	// GRID
		CmdAutCpl					: BOOL; 		(* Coupling authorization	*)
		CmdDisconnect				: BOOL; 		(* Powerplant disconnect order *)
		CmdEmergencyDisconnect		: BOOL; 		(* Powerplant Emergency disconnect order *)
		
	//Project specific ( France ) 
	CmdDisconnect_end			: BOOL; 		(* Powerplant End of disconnect order *)
	CmdEmergencyDisconnect_end	: BOOL; 		(* Powerplant End of Emergency disconnect order *)
	CmdStartPReg				: BOOL ; 		(* Activate P regulation from Grid   *)
	CmdStopPreg                 : BOOL ; 		(* Desactivate P regulation from Grid   *)
	CmdStartQReg                : BOOL ; 		(* Activate Q regulation from Grid   *)
	CmdStopQReg                 : BOOL ; 		(* Desactivate Q regulation from Grid   *)

           	
END_STRUCT
END_TYPE

// ---- 04_Application/OPC/AllDataWToggle.TcDUT
TYPE AllDataWToggle :
STRUCT
	// Toggle command
		CmdStopServer_SMS		: BOOL ;	(* Disable SMS Server *)
		
END_STRUCT
END_TYPE

// ---- 04_Application/OPC/AllValueW.TcDUT
TYPE AllValueW :
STRUCT
 // PP 
	SetptTanPhi_PP				: REAL; 										(* (p.u) TanPhi setpoint to regulate if the corresponding mode is activated *)

// SMS 	
	AX_NbPhone_OPC				: ARRAY[1..CstNbUser] OF STRING(26);			(* List of the phone number to be registered for SMS functions *)
	AX_SubscribedSms_OPC		: ARRAY[1..CstNbUser] OF BOOL;					(* List of subscription for SMS function *)
	AX_NamesUsers_OPC					: ARRAY[1..CstNbUser] OF STRING(50);	(* List of SMS user names *)
	AX_MailAddr_OPC				: ARRAY[1..CstNbUser] OF STRING(255);			(* Contient tous les numéros des utilisateurs *)
	AX_SubscribedMail_OPC		: ARRAY[1..CstNbUser] OF BOOL;					(* List of subscription for MAIL function *)
	AX_UserLVL					: ARRAY[1..CstNbUser] OF WORD;					(* Bit-wise encoding of Alarm subscription (Check Config alarm document for bit signification) *)
	
// SUB	
	SetpP_SUB					: REAL;											(* (kW) Active Power setpoint to be regulated at Subatstion ( if local setpoint enabled) *)
    SetpQ_SUB					: REAL;											(* (kVAr) Reactive Power setpoint to be regulated at Subatstion ( if local setpoint enabled) *)
// PTR 
	SetpP_INV					: ARRAY[1..CstNbPTR_G] OF ARRAY[1..CstNbInv_PTR_G] OF  REAL;	(*(kW) Active Power setpoint to be regulated at the inverter ( if local setpoint enabled) *) 	
	
END_STRUCT
END_TYPE

// ---- 00_FunctionsBlocks/Beckhoff/Communication/IEC104/GVL_Cst.TcGVL
{attribute 'qualified_only'}
VAR_GLOBAL CONSTANT
		CstNbAOEntries			: INT :=  50 ;
END_VAR

// ---- 00_FunctionsBlocks/Beckhoff/Fifo/GVL_Fifo.TcGVL
VAR_GLOBAL CONSTANT 
		Max_buffer_size_G					: UDINT:=10000000; // Max buffer size of fifo
END_VAR

// ---- 04_Application/CONFIG/GVL_BASE.TcGVL
///////////////////////
// DO NOT MODIFY :  
// Maximal number of objects  - Maximal array size 
////////////////////
VAR_GLOBAL CONSTANT 
	// PRODUCT 
	CstNbPTR_G					: BYTE := 4 ;  				// (NA) Number of PTR
	CstNbESS_G   				: BYTE := 3 ;  				// (NA) Number of ESS


// EQUIPMENT
	
	//SUB_MV
	
		CstNbFeederMVCB_G			: BYTE	:= 3 ; 
		CstNbGridMVCB_G				: BYTE	:= 2 ; 
	
	// PTR 
	
		CstNbInv_PTR_G				: BYTE := 5 ;	// Maximal Number of PV Inverters for PTR
		CstNbTempTansfo_PTR_G		: BYTE := 2 ; 	// Maximal Number of Transformer temperature
		CstNbSB_INV_G				: BYTE := 32 ;	// Maximal Number of String box in inverter
		CstNb_DU_G					: BYTE := 2  ;	// Maximal number of DU ? DC inputs ? 
		CstNbPowerCol_INV_G			: BYTE := 3 ; 	// Maximal number of Power Columns per inverter 
		CstNbSB_DcModule_G			: BYTE := 15 ; 	// Maximal number of String box in DC Module 
		CstNbDcModule_INV_G			: BYTE := 15 ;	 // Maximal number of DC Module by inverter
		CstNbSTR_SB_G				: BYTE := 32 ;	// Maximal Number of String by String box 
		
	// EM 
		
		CstNbEM_G					: BYTE := 2;				// Number of Energy Meters
		
	//ESS		
	
		CstNbPcs_ESS_G					: BYTE := 2  ;
		CstNbPowerCol_PCS_G				: BYTE := 6  ;				// Maximal Number of Power colonne by PCS
		CstNbHvac_ESS_G					: BYTE := 2  ;
		CstNbBAT_ESS_G					: BYTE := 2  ;
		CstNbRack_BAT_G					: BYTE := 2  ;
		CstNbModule_Rack_G				: BYTE := 25  ;
		CstNbBms_BAT_G					: BYTE := 1  ;
		CstNbDU_PCS_G					: BYTE := 2  ;
		CstNbTempSensor_ESS_G			: BYTE := 4  ;
		CstNbHygroSensor_ESS_G			: BYTE := 4  ;
		CstNbDS_Ess_G					: BYTE := 2  ;
		CstNbSS_Ess_G					: BYTE := 2  ;
		CstNbEs_ESS_G					: BYTE := 2  ;
		CstNbChainDcSwitchBank_Ess_G	: BYTE := 2  ;	
		
		
	//WS	
	
		CstNbPyrano_GTI				: UINT := 5;
		CstNbPyrano_GHI				: UINT := 5;
		CstNbAnemo					: UINT := 1;
		CstNbPanTmp					: UINT := 4;
		CstNbAmbTmp					: UINT := 3;	
		
	// PP 
	
		CstNbCouplermax_G			: BYTE 	:= 100 ;			// Maximal number of ethercat devices 
		CstNbAlarmIO_G				: BYTE := 10 ; // Number of Event in PRG_IO.
		
	//TRK 
	
		CstNbTrk_NCU_G				: BYTE := 200 ; 
	
	(*               SMS               							*)
	CstNbUser					: SINT:=10; //Nbr d'utilisateur utilisé par AX_Numtel
	CstNbCMD					: SINT:=20; //Nbr commande utilisé par AX_CMD_SMS
	CstNbAlarmCode				: INT:=400;  //Number of alarmcode use in AlarmManager
	
	// TIMEZONE
	    (* Indonesia East Standard Time Zone settings *)
        FRANCE_TZI : ST_TimeZoneInformation := (bias:=-60,
                                       		 				standardName:='Heure Française',
                                        					standardDate:=(wYear:=0,wMonth:=10,wDayOfWeek:=0,wDay:=27,wHour:=3),
                                        					standardBias:=0,
                                        					daylightName:='None',
                                        					daylightDate:=(wYear:=0,wMonth:=3,wDayOfWeek:=0,wDay:=31,wHour:=2),
                                        					daylightBias:=0);
			
		CstPhoneIndicator_G		: STRING := '+33';
			
			CstCycleTime_G		: INT := 10 ; 			// (ms) Cycle Time of the CPU FB Main 
			CstCycleTime_Annex	: INT := 100 ; 			// (ms) Cycle Time of the CPU FB Annex_Function

		CstNbRedundantVariableMax_G	: UINT := 553 ;
		CstNbParamOPCUA				: UINT := 100 ; 
	
END_VAR
VAR_GLOBAL
	sTimeGMT_G          	: STRING;				// Full Date Time for historization (GMT) 
	sTimeLocal_G		 	: STRING ;				// Local Time 
	CalGMTTimeStruct		: TIMESTRUCT ; 			// GMT Time Structure

	ParamOpenVpnFile		: STRING := '';			// Path to openvpn file. 
	ParamIpPublic 			: STRING(255);			// Public IP 
	MesSizeCdrive_PLC		: REAL := 100000 ; 		// (Mo) Remaining Disk space
	MesSizeCdrive_IndusPC	: REAL := 100000 ; 		// (Mo) Remaining Disk space
END_VAR

// ---- 04_Application/CONFIG/GVL_Beckhoff.TcGVL
VAR_GLOBAL
	CalLocalTimeStruct			: TIMESTRUCT;		// Local Time Structure
	CstTimeZone_G				: ST_TimeZoneInformation 	:= WEST_EUROPE_TZI ;	// Local TimeZone
	ParamDirBaseStore		: STRING := 'C:\TwinCAT\Functions\Historisation\';	// Directroy for the historization
	
	
	// Communication 
	stPCComInData  	AT %I*	: EL6inData22B;//PcComInData; 	//DATA qui rentre  ELinData22B;
	stPCComOutData	AT %Q*	: El6outdata22b;//PcComOutData; //DATA qui sort  EL6outData22B;
	stTxBufferPC			: ComBuffer; 	//Connection serie
	stRxBufferPC			: ComBuffer; 	//Connection serie
	
END_VAR

// ---- 04_Application/CONFIG/GVL_CFG.TcGVL
///////////////
// Configuration Files. Define Power Plant sizing and references. 
//////////////
VAR_GLOBAL 
		CstPLCBackup 			: BOOL := FALSE ;  			// TRUE if this PLC is used as a backup . 
		CstNetAmsId_Slave		: STRING(20):= '5.49.202.22.1.1'; //NetAMSId Slave .'5.79.170.90.1.1'
		CstNetAmsId_IndusPC		: STRING(20):= ''; // set '' if no Indus PLC
		//CstIPIEC104			: STRING := '10.101.111.1' ; 
		
		
END_VAR
	
VAR_GLOBAL 
	// Solar Classique //
		A1_PP					: FB_PP  ;  								// MCA Power Plant 
 
	// PRODUCT DEFINITION //
		//PTR 
		AX_PTR 					: ARRAY[1..CstNbPTR_G] OF FB_PTR ; 	 		// Array with AMG products
		
		//SUB_MV
		A1_SUBMV				: FB_SUBMV ;	 					 		// SUB_MV		

		//SUB_HV
		A1_SUBHV				: FB_SUBHV ;	 					 		// SUB_MV		


		
		//WEATHER STATION
		A1_WS					: FB_WS;
		
		//ESS 
		AX_ESS				: ARRAY[1..CstNbESS_G] OF FB_ESS ; 
		
	// GLOBAL VARIABLE //
	
		CmdClearFault_G			: BOOL ; 									// (NA) Clear all permanent faults
		CmdInit_G				: BOOL ; 									// (NA) Global Init Action
		CstIPIEC104				: STRING := '10.111.109.1' ; 		
END_VAR

// ---- 04_Application/CONFIG/GVL_Check.TcGVL
VAR_GLOBAL
	FaultCheck_G : BOOL ; // Test if Fault 
	Fault_Count_G: CTU  ; // Counter 	
	

END_VAR

// ---- 04_Application/CONFIG/GVL_DataBaseStructures.TcGVL
{attribute 'qualified_only'}
VAR_GLOBAL
	AX_StructModbusTCP 	AT %MW112 	: ARRAY[1..10000] OF WORD;
END_VAR

// ---- 04_Application/Annexes_Functions/PRG_AnnexesFunctions.TcPOU
PROGRAM PRG_AnnexesFunctions
VAR_INPUT PERSISTENT
	ParamServiceName_OPCUA			: STRING(255) := 'OPCUA\';	(*OPC UA Folder Name*)
	ParamServiceName_Teamviewer		: STRING(255) := 'Teamviewer\';	(* Teamviewer Folder Name*)	
	ParamServiceName_HMIServer		: STRING(255) := 'HmiServer\';	(*HmiServer Service Name*)	
	ParamServiceName_Telegraf		: STRING(255) := 'Telegraf\';	(* Telegraf Folder Name*)	
END_VAR
VAR_INPUT
	IN_bStartPing				: BOOL;	
    IN_bStart_IP				: BOOL;
    IN_bStart_PLC				: BOOL;

	IN_CmdRestart_OPCUA 		: BOOL;	// OPC UA , Docker , OPEn VPN , Codesys. Push button
	IN_CmdRestart_Teamviewer 	: BOOL;	// OPC UA , Docker , OPEn VPN , Codesys. Push button
	IN_CmdRestart_HMIServer 	: BOOL;	// OPC UA , Docker , OPEn VPN , Codesys. Push button
	IN_CmdRestart_Telegraf 		: BOOL;	// OPC UA , Docker , OPEn VPN , Codesys. Push button

	IN_bStartVpnConnection		: BOOL;
	IN_bStopVpnConnection		: BOOL;
	IN_AdrIP					: STRING(50);
END_VAR

VAR_INPUT PERSISTENT
	ParamRestartTCHour			: WORD := 3;
	ParamRestartTCEnabled		: BOOL ; 
END_VAR

VAR PERSISTENT 
	RestartCounter 				: UINT;
END_VAR

VAR
		bInit					: BOOL := TRUE ; 
		PRG_RestartService		: ARRAY[1..4] OF FB_RestartService ; 
		StartProcess 			: NT_StartProcess;
		CpuUsage				: TC_CpuUsage;
		TON_ALarm				: TON ; // TON to inhibate alarmes during the first secondes after initailization 

		// Restart Twincta
		Step: INT;
		R_Trig_TP_IP			: R_TRIG;
		TC_Restart1				: TC_Restart;	
		TP_GetIPPublic			: TP;

END_VAR
VAR_OUTPUT 
	CPUUsage_PLC				: UDINT ; 
END_VAR

IF bInit THEN
	M_Init();
	///////// 
END_IF




// Get Public IP : 	Auto query every 10 minutes
	FUN_GetPublicIp(
		ParamNetID := CstNetAmsId_IndusPC ,
		IN_DirExe := 'C:\TwinCAT\Functions\Annex_Fonctions\GetPublicIp\',
		IN_CmdStart := IN_bStart_IP OR (CalLocalTimeStruct.wMinute MOD 10 = 0 AND CalLocalTimeStruct.wSecond = 0
	));

// Ping Host 	
//	FUN_PingHost(IN_bStart := IN_bStartPing, IN_PingAdr := IN_AdrIP, IN_DirBatLocation := 'C:\TwinCAT\Functions\Fonction_Com\Ping\');

// CHECK STATES
	// CPU Usage 	
		CpuUsage(NETID := '', Start := CalLocalTimeStruct.wSecond = 0, TMOUT := T#1S);
		CPUUsage_PLC := 	CpuUsage.USAGE ; 
		
	// Check Disk Space = planned task
	// Check Services = planned task
	// Network Scan = planned task
	
	// VPN Management
		FUN_ConnectVPN(IN_CmdStart := IN_bStartVpnConnection, IN_OpenVpnFile := GVL_BASE.ParamOpenVpnFile);
		FUN_DisconnectVPN(IN_CmdStart := IN_bStopVpnConnection);
		

// RESTART SERVICES 
	// Restart OPC UA  	


			PRG_RestartService[1](ParamNetID:='' , IN_Directory := CONCAT(STR1:='C:\TwinCAT\Functions\AnnexFunctions\RestartService\',STR2:= ParamServiceName_OPCUA), Start:= IN_CmdRestart_OPCUA , IN_ServiceName := 'RestartService.exe');
			PRG_RestartService[2](ParamNetID:='' , IN_Directory := CONCAT(STR1:='C:\TwinCAT\Functions\AnnexFunctions\RestartService\',STR2:= ParamServiceName_Teamviewer), Start:= IN_CmdRestart_Teamviewer , IN_ServiceName := 'RestartService.exe');
			PRG_RestartService[3](ParamNetID:='' , IN_Directory := CONCAT(STR1:='C:\TwinCAT\Functions\AnnexFunctions\RestartService\',STR2:= ParamServiceName_HMIServer), Start:= IN_CmdRestart_HMIServer , IN_ServiceName := 'RestartService.exe');
			PRG_RestartService[4](ParamNetID:='' , IN_Directory := CONCAT(STR1:='C:\TwinCAT\Functions\AnnexFunctions\RestartService\',STR2:= ParamServiceName_Telegraf), Start:= IN_CmdRestart_Telegraf , IN_ServiceName := 'RestartService.exe');



	// Restart PLC 	
		PRG_RestartPlc(CmdRestart:= IN_bStart_PLC);
		
	// Restart Twincat at specified date and time to fix EL6614 issue 
		CASE Step OF
			0: //	
				IF CalLocalTimeStruct.wHour = ParamRestartTCHour AND CalLocalTimeStruct.wMinute = 0 AND (CalLocalTimeStruct.wSecond >= 0 AND CalLocalTimeStruct.wSecond <=  5) AND ParamRestartTCEnabled  THEN 
					Step := 1;
				END_IF
			1:
				TC_Restart1(
					RESTART:= TRUE, 
					TMOUT:= T#500MS );
					RestartCounter:=RestartCounter+1;
		END_CASE
	
// ALARMS	
	//Gestion des alarmes sur active configuration --> Alarme inhibées pendant 10s
	TON_ALarm(IN:= MAIN.OUT_CalRunningPLC_IO , PT:= T#10S) ; 

	IF TON_Alarm.Q THEN 
		FUN_Alarms(IN_Directory := ParamDirBaseStore);
	END_IF
	
	FUN_CreateDir_CSV(InDirectory := ParamDirBaseStore);
	FUN_Write_CSV	(InDirectory := ParamDirBaseStore);

	
// Interfaces // 	

ModbusTcp() ; 
//HMI();

METHOD M_Init : BOOL
VAR_INPUT
END_VAR

VAR
	KK: UINT;
	LL: UINT;
END_VAR
	// Add code activation to the alarms
	
	FUN_Alarms_CSV.FIFO.A_Get();
	FUN_Alarms_CSV.FIFO.A_Remove();	
	FUN_Alarms_CSV.FIFO.In.Message := 'Code Activation';
	FUN_Alarms_CSV.FIFO.In.TimeStamp_Act := SYSTEMTIME_TO_STRING(CalLocalTimeStruct);
	FUN_Alarms_CSV.FIFO.A_Add();
	
	InfluxDb_AlarmsManagement.IN_FIFO.A_Get();
	InfluxDb_AlarmsManagement.IN_FIFO.A_Remove();
	InfluxDb_AlarmsManagement.IN_FIFO.In.Message := 'Code Activation';
	InfluxDb_AlarmsManagement.IN_FIFO.In.TimeStamp_Act := SYSTEMTIME_TO_STRING(CalLocalTimeStruct);
	InfluxDb_AlarmsManagement.IN_FIFO.A_Add();	
	
	FUN_SendMail.FIFO.A_Get();
	FUN_SendMail.FIFO.A_Remove();
	FUN_SendMail.FIFO.In.Message := 'Code Activation';
	FUN_SendMail.FIFO.In.TimeStamp_Act := SYSTEMTIME_TO_STRING(CalLocalTimeStruct);
	FUN_SendMail.FIFO.A_Add();
	
	// Reinitialize all Alarms values 
	FOR KK := 1 TO CstNbAlarmCode DO
		FUN_Alarms.AX_MesAlarmCode[KK] := 0 ; 
		FOR LL:=0 TO 15 DO 
			FUN_Alarms.AX_Journal[KK][LL].Value := FALSE ;
		END_FOR 
	END_FOR
	
	bInit:= False ;
END_METHOD

END_PROGRAM

// ---- 04_Application/OPC/OpcUa.TcPOU
PROGRAM OpcUa
///////////////////
// OPC UA Management 
// Commands are resetted to FALSE right after being received . Protection against rapide consecutives commands . Protection against simultaneous commands.
///////////////////
VAR_INPUT PERSISTENT
	ParamTimeOutTc			: TIME:=T#1S;		(* (s)Minimum duration before two consecutives commands *)
	ParamNbCmdBlock			: UINT  := 1 ; 		(* Number of commands per block. Commands in the same block can not be executed in the same time. *)
//Test
END_VAR             		
                    		
                    		
VAR_INPUT           		
                    		
    {attribute 'OPC.UA.DA' := '1'}                		
	AllDataR 				: AllDataR; // All Data Read Only
	
	{attribute 'OPC.UA.DA' := '1'}                		
	AllDataWPulse 			: AllDataWPulse; //  All boolean OPC UA to be written  that will be converted to tap by resetting the entry to false after two seconds. 
	
	AllDataWToggle 			: AllDataWToggle; // All boolean OPC UA to be written as a toggle
    
    {attribute 'OPC.UA.DA' := '1'}            		
	AllValueW 				: AllValueW; // All non boolean OPC UA data to be  written 
	                		
	AllRtc					: AllDataWPulse;	// OUtput of the AllDataWPulse . 
	
	
	{attribute 'OPC.UA.DA' := '1'}         	
	AllAlarms 	: AllAlarms; // All Alarms Read Only
	
	
	
	// Test Mise à jour Parameters via OPC UA
	
	//AllDataParameterWrite	: AllDataParameter;	// Structure qui permet d'écrire les valeurs des paramètres via OPC UA
   		
END_VAR             		
VAR                 		
//	Buffer_AllW				: ARRAY[1..500] OF BOOL ;      
	Buffer_TcWord			: ARRAY[1..500] OF BOOL ;  
	Buffer_Rtc   			: ARRAY[1..500] OF BOOL ;  
	
	CP_TcAllow				: BOOL; // The power plan can received TC

	bInit					: BOOL;
	TempoTcRunning			: TON;
	                		
	// M_TC //      		
	TcIsRunning				: BOOL;
	NbTcAskedBlock			: BYTE;	    
	bTooManyCmd				: BOOL;		// At least one block has too many simultaneous commands. 
	bAtLeastOne				: BOOL;     // There is at least one commAND                              
	       
	// Force Alarms
	R_TRIG_DisableSMSForceAlarms	: R_TRIG;
	F_TRIG_DisableSMSForceAlarms	: F_TRIG;


                 
	// M_ACKNOWLEDGE        
	F_Tap_OPC						: ARRAY[1..24] OF FB_TapVariable ; 
	F_Tap_OPC_SUB_MV				: ARRAY[1..16] OF FB_TapVariable ; 
	F_Tap_OPC_PTR					: ARRAY[1..CstNbPTR_G] OF ARRAY[1..6] OF FB_TapVariable ;		
	F_Tap_OPC_Inv					: ARRAY[1..CstNbPTR_G] OF ARRAY[1..CstNbInv_PTR_G] OF ARRAY[1..4] OF FB_TapVariable ;		
	F_Tap_OPC_GRID					: ARRAY[1..10] OF FB_TapVariable ; 
	F_Tap_OPC_ESS					: ARRAY[1..10] OF FB_TapVariable ; 
	F_Tap_OPC_PP					: ARRAY[1..10] OF FB_TapVariable ;	
	F_Tap_OPC_SUB_MV_InhibRead		: ARRAY[1..10] OF FB_TapVariable ;	
	
	F_Tap_OPC_INV_InhibRead : ARRAY[1..CstNbPTR_G] OF ARRAY[1..CstNbInv_PTR_G] OF FB_TapVariable ;	
	F_Tap_OPC_SL_InhibRead : ARRAY[1..CstNbPTR_G] OF FB_TapVariable ;	

	F_Tap_Inhib : ARRAY[1..1000] OF FB_TapVariable ;	
	
	
	Test_SmS_Rtrig			: R_TRIG ; 
	Rtrig_StayConnect		: R_TRIG;
	Rtrig_IpLauncher		: R_TRIG;
	Rtrig_HHCollector		: R_TRIG;
	Rtrig_RestartPlc		: R_TRIG;
	R_TRIGTanPhi			: R_TRIG ; 
	R_TRIG_InhibIO			: R_TRIG;
	bReadFromTargetInfos	: BOOL ; 
	// Intermediary commands
	PP_SetptP_Old							: REAL;
	PP_SetptQ_Old							: REAL;
	

	
END_VAR


VAR
	// WAGO Variable transcription
	OpcUaServer_1 : REAL ; 
	OpcUaServer_2 : REAL ; 
	OpcUaServer_3 : REAL ; 
	OpcUaServer_4 : REAL ; 
	OpcUaServer_5 : REAL ; 
	OpcUaServer_6 : REAL ; 
	OpcUaServer_7 : REAL ; 
	OpcUaServer_8 : REAL ; 
	OpcUaServer_9 : REAL ; 
	OpcUaServer_10 : REAL ; 
	OpcUaServer_11 : REAL ; 
	OpcUaServer_12 : REAL ; 
	OpcUaServer_13 : REAL ; 
	OpcUaServer_14 : REAL ; 
	OpcUaServer_15 : REAL ; 
	OpcUaServer_16 : REAL ; 
	OpcUaServer_17 : REAL ; 
	OpcUaServer_18 : REAL ; 
	OpcUaServer_19 : REAL ; 
	OpcUaServer_20 : REAL ; 
	OpcUaServer_21 : REAL ; 
	OpcUaServer_22 : REAL ; 
	OpcUaServer_23 : REAL ; 
	OpcUaServer_24 : REAL ; 
	OpcUaServer_25 : REAL ; 
	OpcUaServer_26 : REAL ; 
	OpcUaServer_27 : REAL ; 
	OpcUaServer_28 : REAL ; 
	OpcUaServer_29 : REAL ; 
	OpcUaServer_30 : REAL ; 
	OpcUaServer_31 : REAL ; 
	OpcUaServer_32 : REAL ; 
	OpcUaServer_33 : REAL ; 
	OpcUaServer_34 : REAL ; 
	OpcUaServer_35 : REAL ; 
	OpcUaServer_36 : REAL ; 
	OpcUaServer_37 : REAL ; 
	OpcUaServer_38 : REAL ; 
	OpcUaServer_39 : REAL ; 
	OpcUaServer_40 : REAL ; 
	OpcUaServer_41 : REAL ; 
	OpcUaServer_42 : REAL ; 
	OpcUaServer_43 : REAL ; 

END_VAR

	IF NOT bInit THEN
		M_Init() ; 
		bInit		:= TRUE ; 
	ELSE
		CP_TcAllow := TRUE;
		M_AlarmManagement() ; 
		M_Evaluate();
		M_TC();
		M_Acknowledge();
		M_InhibAllowAll() ; 
		//M_Wago()
	END_IF

METHOD M_Acknowledge : BOOL
VAR
		KK: INT;
		LL: INT;
	JJ: UINT;
	TapTrigger: BOOL;
	bResetSD : BOOL;
END_VAR


// 					ATTENTION				//
// Utiliser le AllRtc et pas le AllDataR 	//

	
// Defaults Actions
	// Reset SMS Server
	F_Tap_OPC[2](TapTrigger:= AllRtc.CmdReset_ServerSMS , TapOut := SMS_Server.IN_Reset_SmsServer) ; 
	// Delete all SMS
	F_Tap_OPC[3](TapTrigger:= AllRtc.CmdDeleteAllSms , TapOut := SMS_Server.IN_CmdDeleteAllSms) ; 
	// Update SMS & Mail Informations
	F_Tap_OPC[4](TapTrigger:= AllRtc.CmdChangeInfos_PhoneEmail , TapOut := SMS_Server.IN_ChangePhoneMailInfos_OPC) ; 
	F_Tap_OPC[5](TapTrigger:= AllRtc.CmdChangeInfos_PhoneEmail , TapOut := FUN_SendMail.IN_ChangePhoneMailInfos_OPC) ; 
	bReadFromTargetInfos :=	AllRtc.CmdReadInfosFromTarget_PhoneEmail ; 
	// Collect Ip Public
	Rtrig_IpLauncher(CLK:=AllRtc.CmdIpLauncher);
	F_Tap_OPC[6](TapTrigger:= Rtrig_IpLauncher.Q , TapOut := PRG_AnnexesFunctions.IN_bStart_IP) ; 
	
	// Toogle Forced Connect
	Rtrig_StayConnect(CLK:=AllRtc.CmdForcedStay_Connect);
	IF Rtrig_StayConnect.Q THEN
		A1_PP.ParamForcedStayConnect := NOT	A1_PP.ParamForcedStayConnect ;
	END_IF
	// Restart PLC
	//Rtrig_RestartPlc(CLK:=AllRtc.CmdRestart_PLC);
	F_Tap_OPC[8](TapTrigger:= AllRtc.CmdRestart_PLC , TapOut := PRG_AnnexesFunctions.IN_bStart_PLC) ; 
	// Restart Routeur ADSL
	F_Tap_OPC[9](TapTrigger:= AllRtc.CmdReset_Router_ADSL, TapOut := A1_SUBMV.A1_Router_ADSL.IN_CmdRestart) ; 
	//Reset MailServer
	F_Tap_OPC[10](TapTrigger:= AllRtc.CmdReset_ServerMail, TapOut := FUN_SendMail.IN_Reset_OPC) ; 
	// Test sms
	A1_PP.IN_TestMailSms	:=	AllRtc.CmdTestSms;
	
	// Restart Routeur 4G
	F_Tap_OPC[12](TapTrigger:= AllRtc.CmdReset_Router_4G, TapOut := A1_SUBMV.A1_Router_4G.IN_CmdRestart) ;
 	// Restart IPC
	F_Tap_OPC[13](TapTrigger:= AllRtc.CmdReset_IPC, TapOut := A1_SUBMV.A1_IPC.IN_CmdRestart) ;
	
	// Disable sms serveur
	F_Tap_OPC[14](TapTrigger:= AllDataWToggle.CmdStopServer_SMS, TapOut := FUN_Alarms.ParamDisableSMS) ; 
	// Start VPN
	F_Tap_OPC[15](TapTrigger:= AllRtc.CmdStart_Vpn, TapOut := PRG_AnnexesFunctions.IN_bStartVpnConnection) ; 
	// Stop VPN
	F_Tap_OPC[16](TapTrigger:= AllRtc.CmdStop_Vpn, TapOut := PRG_AnnexesFunctions.IN_bStopVpnConnection) ;

	
	
	// Restart Services
	F_Tap_OPC[18](TapTrigger:= AllRtc.CmdRestart_OPCUA 		 , TapOut := PRG_AnnexesFunctions.IN_CmdRestart_OPCUA) ; // 
	F_Tap_OPC[20](TapTrigger:= AllRtc.CmdRestart_Teamviewer	 , TapOut := PRG_AnnexesFunctions.IN_CmdRestart_Teamviewer) ; // 
	F_Tap_OPC[21](TapTrigger:= AllRtc.CmdRestart_HMIServer 	 , TapOut := PRG_AnnexesFunctions.IN_CmdRestart_HMIServer ) ; // 
	F_Tap_OPC[23](TapTrigger:= AllRtc.CmdRestart_Telegraf 	 , TapOut := PRG_AnnexesFunctions.IN_CmdRestart_Telegraf 	 ) ; // 		
			
	F_Tap_OPC[24](TapTrigger:= AllRtc.CmdReset_SD		 	, TapOut := bResetSD 	 ) ; // 		
		
	IF bResetSD THEN
		//A1_SUBMV.A1_SD_LV.IN_CmdReset_L := bResetSD;
		A1_SUBMV.A1_SD_MV.IN_CmdReset_L := bResetSD;
		FOR KK := 1 TO CstNbPTR_G DO 
			AX_PTR[KK].A1_SD_INV.IN_CmdReset_L 		:= bResetSD;
			AX_PTR[KK].A1_SD_Transfo.IN_CmdReset_L 	:= bResetSD;
			
		END_FOR
	END_IF

//SUB_MV
	F_Tap_OPC_SUB_MV[1](TapTrigger:= AllRtc.CmdOpen_MainMVCB , TapOut 	:= A1_SUBMV.IN_CmdOpenMainMVCB) ; 
	F_Tap_OPC_SUB_MV[2](TapTrigger:= AllRtc.CmdClose_MainMVCB , TapOut 	:= A1_SUBMV.IN_CmdCloseMainMVCB) ;
	F_Tap_OPC_SUB_MV[3](TapTrigger:= AllRtc.CmdReset_MainMVCB , TapOut 	:= A1_SUBMV.A1_MainMVCB.IN_CmdReset) ; 
	F_Tap_OPC_SUB_MV[4](TapTrigger:= AllRtc.CmdRestart_UPS48 , TapOut 	:= A1_SUBMV.A1_UPS_48v.IN_CmdReStartUPS) ;
	F_Tap_OPC_SUB_MV[4](TapTrigger:= AllRtc.CmdRestart_UPS24 , TapOut 	:= A1_SUBMV.A1_UPS_24v.IN_CmdReStartUPS) ;  	
	
	FOR KK:= 1 TO CstNbFeederMVCB_G DO 
		F_Tap_OPC_SUB_MV[4+(KK-1)*3+1](TapTrigger:= AllRtc.CmdOpen_FeederMVCB[KK] , TapOut := A1_SUBMV.IN_CmdOpenFeederMVCB[KK]) ; 
		F_Tap_OPC_SUB_MV[4+(KK-1)*3+2](TapTrigger:= AllRtc.CmdClose_FeederMVCB[KK] , TapOut := A1_SUBMV.IN_CmdCloseFeederMVCB[KK]) ; 
		F_Tap_OPC_SUB_MV[4+(KK-1)*3+3](TapTrigger:= AllRtc.CmdReset_FeederMVCB[KK] , TapOut := A1_SUBMV.AX_FeederMVCB[KK].IN_CmdReset) ; 

		
	END_FOR 	
	
// PTR 
FOR KK := 1 TO UINT_TO_INT(CstNbPTR_G) DO
	F_Tap_OPC_PTR[KK][1](TapTrigger:= AllRtc.CmdClose_PTR[KK] , TapOut := AX_PTR[KK].A1_MainMVCB_PTR.IN_CmdClose) ;
	F_Tap_OPC_PTR[KK][2](TapTrigger:= AllRtc.CmdOpen_PTR[KK] , TapOut := AX_PTR[KK].A1_MainMVCB_PTR.IN_CmdOpen) ;
	
	FOR JJ:=1 TO CstNbInv_PTR_G DO 
		F_Tap_OPC_Inv[KK][JJ][1](TapTrigger:= AllRtc.CmdStop_INV[KK][JJ] , TapOut := AX_PTR[KK].AX_INV[JJ].IN_CmdStop_Local ) ;
		F_Tap_OPC_Inv[KK][JJ][2](TapTrigger:= AllRtc.CmdStart_INV[KK][JJ] , TapOut := AX_PTR[KK].AX_INV[JJ].IN_CmdStart_Local ) ;		
		
		F_Tap_OPC_Inv[KK][JJ][3](TapTrigger:= AllRtc.CmdToggleCom_Read[KK][JJ] , TapOut := AX_PTR[KK].AX_INV[JJ].IN_CmdToggleRead ) ;
		F_Tap_OPC_Inv[KK][JJ][4](TapTrigger:= AllRtc.CmdToggleCom_Write[KK][JJ] , TapOut := AX_PTR[KK].AX_INV[JJ].IN_CmdToggleWrite ) ;		
	
		IF AllRtc.CmdStartSetptP_INV[KK][JJ] THEN 
			AX_PTR[KK].AX_INV[JJ].IN_SetptPlimit_Local :=  AllValueW.SetpP_INV[KK][JJ] ; 
		END_IF
		IF AllRtc.CmdStopSetptP_INV[KK][JJ] THEN 
			AX_PTR[KK].AX_INV[JJ].IN_SetptPlimit_Local :=  AX_PTR[KK].AX_INV[JJ].ParamPn ; 
		END_IF
		
	END_FOR
	

	

END_FOR

// DEIE
	F_Tap_OPC_GRID[1](TapTrigger:= AllRtc.CmdAutCpl , TapOut := A1_SUBMV.A1_GRID.IN_CmdAutCpl_other) ; 
	F_Tap_OPC_GRID[2](TapTrigger:= AllRtc.CmdDisconnect , TapOut := A1_SUBMV.A1_GRID.IN_CmdDisconnect_other) ; 
	F_Tap_OPC_GRID[3](TapTrigger:= AllRtc.CmdDisconnect_end , TapOut := A1_SUBMV.A1_GRID.IN_CmdDisconnect_end_other) ; 
	F_Tap_OPC_GRID[4](TapTrigger:= AllRtc.CmdEmergencyDisconnect , TapOut := A1_SUBMV.A1_GRID.IN_CmdEmergencyDisconnect_other) ; 	
	F_Tap_OPC_GRID[5](TapTrigger:= AllRtc.CmdEmergencyDisconnect_end , TapOut := A1_SUBMV.A1_GRID.IN_CmdEmergencyDisconnect_End_other) ; 	
	F_Tap_OPC_GRID[6](TapTrigger:= AllRtc.CmdStartPReg 		, TapOut := A1_SUBMV.A1_GRID.IN_CmdStartPReg_other) ; 
	F_Tap_OPC_GRID[7](TapTrigger:= AllRtc.CmdStopPReg 		, TapOut := A1_SUBMV.A1_GRID.IN_CmdStopPReg_other) ; 
	F_Tap_OPC_GRID[8](TapTrigger:= AllRtc.CmdStartQReg 		, TapOut := A1_SUBMV.A1_GRID.IN_CmdStartQReg_other) ; 
	F_Tap_OPC_GRID[9](TapTrigger:= AllRtc.CmdStopQReg 		, TapOut := A1_SUBMV.A1_GRID.IN_CmdStopQReg_other) ; 


//SUB_MV
	IF AllRtc.CmdStartLocalSetptP_PP THEN
		A1_PP.IN_PIDP_SetptP_local			:=	AllValueW.SetpP_SUB;
		A1_PP.IN_CmdPIDP_LocalMode 	:= TRUE;
	END_IF
	
	IF AllRtc.CmdStopLocalSetptP_PP THEN
		A1_PP.IN_CmdPIDP_LocalMode  	:= FALSE; 
		A1_PP.IN_PIDP_SetptP_local		:= A1_PP.ParamPmax;               
	END_IF
	
// ESS
	F_Tap_OPC_ESS[1](TapTrigger := AllRtc.CmdCloseDc_BAT[1][1], TapOut := AX_ESS[1].AX_Bat[1].IN_CmdCloseDC);
	F_Tap_OPC_ESS[2](TapTrigger := AllRtc.CmdCloseDc_BAT[1][2], TapOut := AX_ESS[1].AX_Bat[2].IN_CmdCloseDC);
	F_Tap_OPC_ESS[3](TapTrigger := AllRtc.CmdOpenDc_BAT[1][1], 	TapOut := AX_ESS[1].AX_Bat[1].IN_CmdOpenDC);
	F_Tap_OPC_ESS[4](TapTrigger := AllRtc.CmdOpenDc_BAT[1][2], 	TapOut := AX_ESS[1].AX_Bat[2].IN_CmdOpenDC);
	F_Tap_OPC_ESS[5](TapTrigger := AllRtc.CmdStart_PCS[1][1], 	TapOut := AX_ESS[1].AX_PCS[1].IN_CmdStart);
	F_Tap_OPC_ESS[6](TapTrigger := AllRtc.CmdStop_PCS[1][1], 	TapOut := AX_ESS[1].AX_PCS[1].IN_CmdStop);
	F_Tap_OPC_ESS[7](TapTrigger := AllRtc.CmdStandby_PCS[1][1], TapOut := AX_ESS[1].AX_PCS[1].IN_CmdStandby);
	F_Tap_OPC_ESS[8](TapTrigger := AllRtc.CmdLocal_PCS[1][1], 	TapOut := AX_ESS[1].AX_PCS[1].IN_CmdPcsInLocalMode);
	F_Tap_OPC_ESS[9](TapTrigger := AllRtc.CmdReset_PCS[1][1], 	TapOut := AX_ESS[1].AX_PCS[1].IN_CmdReset);
	
// PP 
	R_TRIGTanPhi(CLK:= AllRtc.CmdWriteSetptTanPhi ) ; 
	IF R_TRIGTanPhi.Q THEN 
		A1_PP.Param_SetptTanPhi  :=  AllValueW.SetptTanPhi_PP ; 		
	END_IF


//MAIL - SMS 
IF bReadFromTargetInfos THEN 
	AllValueW.AX_MailAddr_OPC		 := AllDataR.MAIL.AX_MailAddr   ; 
	AllValueW.AX_NamesUsers_OPC 	 := AllDataR.MAIL.AX_NomUtili 	; 
	AllValueW.AX_NbPhone_OPC		 := AllDataR.SMS.AX_Numtel 		; 	
	AllValueW.AX_SubscribedMail_OPC  := AllDataR.MAIL.AX_Subscribed ; 	
	AllValueW.AX_SubscribedSms_OPC   := AllDataR.SMS.AX_Subscribed  ; 	
	AllValueW.AX_UserLVL 			 := AllDataR.MAIL.AX_UserLVL    ;  		
	
	bReadFromTargetInfos 			 := FALSE ;
END_IF
END_METHOD

METHOD M_AlarmManagement
//////////////////
// Generates object alarms and manages resets. 
//////////////////

VAR 
	// Method local variables (reinitialized at each cycle) 
	FB_AlarmCodeManager			: FB_AlarmCodeManager ;

	TransfoAlarmCode			: WORD;
	TransfoWarningCode			: WORD;
	ANATempWarningCode			: WORD;    // ANA Temperature Warning Code synthesis 
	ANATempAlarmCode			: WORD;    // ANA Temperature Alarm Code synthesis                               

	AlarmCodeSD_Transfo			: WORD;    // Sd Alarm Code synthesis PTR
	AlarmCodeSD_INV				: WORD;    // Sd Alarm Code synthesis SCADA
	
	VaneWarningCode             : WORD;
	TempSensor_Amb_1WarningCode	: WORD;
	TempSensor_Amb_2WarningCode	: WORD;
	TempSensor_TransfoWarningCode: WORD;

	InvComWarning				: BOOL;		// Aggregated communication warning
	InvComError					: BOOL;		// Aggregated communication Alarm
	InvAlarmCode				: WORD; 
	InvWarningcode				: WORD;
	
	DS_Transfo					: BOOL;
	DS_INV						: BOOL;
END_VAR

	
// ALARM CODE //

// Attention une alarm doit être mise en commentaire de la manière suivante (* *), l'utilisation du // pose pb sur Bazefield 

	FB_AlarmCodeManager(
		bAlarm1			:= FALSE,//
		bAlarm2			:= FALSE,//
		bAlarm3			:= FALSE,//
		bAlarm4			:= FALSE,//
		bAlarm5			:= FALSE,//
		bAlarm6			:= FALSE,//
		bAlarm7			:= FALSE,//
		bAlarm8			:= FALSE,//
		bAlarm9			:= FALSE,//
		bAlarm10		:= FALSE,//
		bAlarm11		:= FALSE,//
		bAlarm12		:= FALSE,//
		bAlarm13		:= FALSE,//
		bAlarm14		:= FALSE,//
		bAlarm15		:= FALSE,//
		wAlarmCode		=> AllDataR.OPCUA.MesAlarmCode);

// WARNING CODE //
	FB_AlarmCodeManager(
 		bAlarm1			:= CP_TcAllow AND bTooManyCmd AND NOT   TcIsRunning,	// two many action in the same time requested                                 
		bAlarm2			:= bAtLeastOne AND  NOT bTooManyCmd AND NOT CP_TcAllow,  					// Cmd send but the PP do not allow TC
		bAlarm3			:= CP_TcAllow AND bAtLeastOne AND  NOT bTooManyCmd AND   TcIsRunning,		// Wait for previous command to be executed.
		bAlarm4			:= FALSE,//
		bAlarm5			:= FALSE,//
		bAlarm6			:= FALSE,//
		bAlarm7			:= FALSE,//
		bAlarm8			:= FALSE,//
		bAlarm9			:= FALSE,//
		bAlarm10		:= FALSE,//
		bAlarm11		:= FALSE,//
		bAlarm12		:= FALSE,//
		bAlarm13		:= FALSE,//
		bAlarm14		:= FALSE,//
        bAlarm15		:= FALSE,//
		wAlarmCode		=> AllDataR.OPCUA.MesWarningCode);
FB_AlarmCodeManager(
bAlarm1         :=allDataWPulse.CmdReset_ServerSMS,//Reset SMS Server #Interface
bAlarm2         :=allDataWPulse.CmdReset_ServerMail,//Reset Mail server #Interface
bAlarm3         :=allDataWPulse.CmdReset_Router_ADSL,//Restart ADSL router #Interface
bAlarm4         :=allDataWPulse.CmdReset_Router_4G,//Restart 4G router #Interface
bAlarm5         :=allDataWPulse.CmdReset_IPC,//Restart IPC #Interface
bAlarm6         :=allDataWPulse.CmdDeleteAllSms,//Delete all SMS in the buffer #Interface
bAlarm7         :=allDataWPulse.CmdChangeInfos_PhoneEmail,//Apply new changes in MAil and SMS infos #Interface
bAlarm8         :=allDataWPulse.CmdReadInfosFromTarget_PhoneEmail,//Get Saved configuration #Interface
bAlarm9         :=allDataWPulse.CmdTestSms,//Test SMS function #Interface
bAlarm10         :=FALSE,
bAlarm11         :=allDataWPulse.CmdRestart_OPCUA,//Restart OPCUA #Interface
bAlarm12         :=FALSE,
bAlarm13         :=allDataWPulse.CmdRestart_Teamviewer,//Restart Teamviewer #Interface
bAlarm14         :=allDataWPulse.CmdRestart_HMIServer,//Restart HMIServer #Interface
bAlarm15         :=FALSE,
wAlarmCode      => AllDataR.OPCUA.MesEventCode[1]);
END_METHOD

METHOD M_Evaluate : BOOL
VAR_INPUT
END_VAR


VAR
	KK: UINT;
END_VAR

AllDataR.PP			:=  A1_PP.MesData ; 
AllDataR.SUBMV	    :=  A1_SUBMV.MesDataExd; 
AllDataR.SUBHV		:= A1_SUBHV.MesDataExd ;

FOR KK:=1 TO CstNbPTR_G DO
	AllDataR.PTR[KK]	    :=  AX_PTR[KK].MesDataExd;
END_FOR

FOR KK:=1 TO CstNbESS_G DO
	AllDataR.ESS_Test[KK]	    :=  AX_ESS[KK].MesDataExd;
	AllDataR.ESS[KK]	    :=  AX_ESS[KK].MesDataExd;

END_FOR



AllDataR.WS	        :=  A1_WS.MesDataExd; 

AllDataR.SMS	    :=  SMS_Server.MesData;
AllDataR.MAIL       :=  FUN_SendMail.MesData;

AllDataR.CSV		:= FUN_Alarms_CSV.MesData; 
AllDataR.CSVData := FUN_Write_CSV.WriteValue.MesData ; 
AllDataR.IO		:= PRG_IO.MesData ; 

R_TRIG_DisableSMSForceAlarms(CLK := FUN_Alarms.bTestForceAlarms);	
F_TRIG_DisableSMSForceAlarms(CLK := FUN_Alarms.bTestForceAlarms);	
	
IF R_TRIG_DisableSMSForceAlarms.Q THEN	
	FUN_Alarms.ParamDisableSMS := TRUE;
	FUN_Alarms.bTriggerCount := TRUE;
	
END_IF	
	
IF F_TRIG_DisableSMSForceAlarms.Q THEN	
	FUN_Alarms.ParamDisableSMS := FALSE;
	FUN_Alarms.MesAlarmWordTestJulienDecouple[FUN_Alarms.nCountSequence-1] := 0 ;  // reinitialize last alarm
	FUN_Alarms.nCountSequence := 0;
	FUN_Alarms.bTriggerCount := FALSE;
END_IF	
	
IF FUN_Alarms.bTestForceAlarms THEN	
	FUN_Alarms.M_ForceAlarms();
END_IF	
	
M_EvaluateAlarms();
END_METHOD

METHOD M_EvaluateAlarms  : BOOL
VAR_INPUT
END_VAR

VAR
	aa: INT;
END_VAR
IF FUN_Alarms.bTestForceAlarms THEN
OpcUa.AllDataR.PP.MesAlarmCode:= A1_PP.MesData.MesAlarmCode; 
OpcUa.AllDataR.PP.MesWarningCode:= A1_PP.MesData.MesWarningCode; 
OpcUa.AllDataR.PP.MesWarningCode2:= A1_PP.MesData.MesWarningCode2; 
OpcUa.AllDataR.PP.MesEventCode:= A1_PP.MesData.MesEventCode; 

	
END_IF
AllAlarms.PP_MesAlarmCode_1:=OpcUa.AllDataR.PP.MesAlarmCode.1;
AllAlarms.PP_MesAlarmCode_2:=OpcUa.AllDataR.PP.MesAlarmCode.2;
AllAlarms.PP_MesAlarmCode_3:=OpcUa.AllDataR.PP.MesAlarmCode.3;
AllAlarms.PP_MesAlarmCode_4:=OpcUa.AllDataR.PP.MesAlarmCode.4;
AllAlarms.PP_MesAlarmCode_5:=OpcUa.AllDataR.PP.MesAlarmCode.5;
AllAlarms.PP_MesWarningCode_1:=OpcUa.AllDataR.PP.MesWarningCode.1;
AllAlarms.PP_MesWarningCode_2:=OpcUa.AllDataR.PP.MesWarningCode.2;
AllAlarms.PP_MesWarningCode_3:=OpcUa.AllDataR.PP.MesWarningCode.3;
AllAlarms.PP_MesWarningCode_5:=OpcUa.AllDataR.PP.MesWarningCode.5;
AllAlarms.PP_MesWarningCode_6:=OpcUa.AllDataR.PP.MesWarningCode.6;
AllAlarms.PP_MesWarningCode_7:=OpcUa.AllDataR.PP.MesWarningCode.7;
AllAlarms.PP_MesWarningCode_8:=OpcUa.AllDataR.PP.MesWarningCode.8;
AllAlarms.PP_MesWarningCode_9:=OpcUa.AllDataR.PP.MesWarningCode.9;
AllAlarms.PP_MesWarningCode_10:=OpcUa.AllDataR.PP.MesWarningCode.10;
AllAlarms.PP_MesWarningCode_12:=OpcUa.AllDataR.PP.MesWarningCode.12;
AllAlarms.PP_MesWarningCode_13:=OpcUa.AllDataR.PP.MesWarningCode.13;
AllAlarms.PP_MesWarningCode_14:=OpcUa.AllDataR.PP.MesWarningCode.14;
AllAlarms.PP_MesWarningCode_15:=OpcUa.AllDataR.PP.MesWarningCode.15;
AllAlarms.PP_MesWarningCode2_1:=OpcUa.AllDataR.PP.MesWarningCode2.1;
AllAlarms.PP_MesWarningCode2_2:=OpcUa.AllDataR.PP.MesWarningCode2.2;
AllAlarms.PP_MesWarningCode2_3:=OpcUa.AllDataR.PP.MesWarningCode2.3;
AllAlarms.PP_MesWarningCode2_4:=OpcUa.AllDataR.PP.MesWarningCode2.4;
AllAlarms.PP_MesWarningCode2_6:=OpcUa.AllDataR.PP.MesWarningCode2.6;
AllAlarms.PP_MesWarningCode2_7:=OpcUa.AllDataR.PP.MesWarningCode2.7;
AllAlarms.PP_MesWarningCode2_8:=OpcUa.AllDataR.PP.MesWarningCode2.8;
AllAlarms.PP_MesWarningCode2_9:=OpcUa.AllDataR.PP.MesWarningCode2.9;
AllAlarms.PP_MesWarningCode2_10:=OpcUa.AllDataR.PP.MesWarningCode2.10;
AllAlarms.PP_MesWarningCode2_11:=OpcUa.AllDataR.PP.MesWarningCode2.11;
AllAlarms.PP_MesWarningCode2_12:=OpcUa.AllDataR.PP.MesWarningCode2.12;
AllAlarms.PP_MesWarningCode2_14:=OpcUa.AllDataR.PP.MesWarningCode2.14;
AllAlarms.PP_MesEventCode_14:=OpcUa.AllDataR.PP.MesEventCode.14;
AllAlarms.PP_MesEventCode_15:=OpcUa.AllDataR.PP.MesEventCode.15;
END_METHOD

METHOD M_InhibAllowAll : BOOL
VAR
		KK: INT;
		LL: INT;
	JJ: UINT;
	TapTrigger: BOOL;
END_VAR


// 					ATTENTION				//
// Utiliser le AllRtc et pas le AllDataR 	//
END_METHOD

METHOD M_Init : BOOL
VAR_INPUT
END_VAR
																
//AllDataWPulse.CmdInhibAllWrite := TRUE  	;
END_METHOD

METHOD M_TC : BOOL
VAR_INPUT
END_VAR

VAR
	AllDataW_0 				: AllDataWPulse; // All Data Write
	KK						: UINT;
	BlockElemCount			: UINT;	// Current element in current block.

END_VAR
MEMCPY(srcAddr := ADR(AllDataWPulse) ,destAddr:= ADR(Buffer_TcWord) ,n:= SIZEOF(AllDataWPulse) ) ; 

NbTcAskedBlock	:= 0;
TcIsRunning		:= FALSE ; 
BlockElemCount 	:=1 ;
bTooManyCmd 	:= FALSE ; 
bAtLeastOne		:= FALSE ;

FOR KK:=1 TO SIZEOF(AllDataWPulse) DO 
	
	IF Buffer_TcWord[KK] THEN // la commande est à True . 
		NbTcAskedBlock := NbTcAskedBlock + 1 ; 
	END_IF
	
	IF Buffer_Rtc[KK] THEN // une commande est en cours 
		TcIsRunning:= TRUE   ;
	END_IF	
	
	IF ParamNbCmdBlock <= BlockElemCount THEN // Fin d'un block. On regarde si il y a eu une commande mais pas plusieurs. 
		BlockElemCount := 1 ; 
		bTooManyCmd	:=bTooManyCmd  OR  NbTcAskedBlock>1 ; 
		bAtLeastOne :=bAtLeastOne  OR NbTcAskedBlock=1; 
		NbTcAskedBlock := 0 ;
		
	ELSE
		BlockElemCount :=  BlockElemCount + 1 ;
	END_IF
END_FOR
// To consider last block
bAtLeastOne := bAtLeastOne OR  NbTcAskedBlock=1; 	
bTooManyCmd	:= bTooManyCmd OR  NbTcAskedBlock>1 ; 

IF CP_TcAllow AND bAtLeastOne AND NOT bTooManyCmd AND NOT TcIsRunning THEN 	// On ne process les commandes que si aucun block n'a pas de double commande, mais qu'au moins un en a une. 
	Buffer_Rtc := Buffer_TcWord  ; 
END_IF

MEMCPY(srcAddr := ADR(Buffer_Rtc) ,destAddr:= ADR(AllRtc) ,n:= SIZEOF(AllRtc) ) ; 

IF bAtLeastOne OR bTooManyCmd THEN 
	//Reset at each cycle
	AllDataWPulse := AllDataW_0;
END_IF


//SECURITY
	TempoTcRunning(IN:= TcIsRunning AND CP_TcAllow , PT:=ParamTimeOutTc);
	
	IF TempoTcRunning.Q THEN
		AllRtc 	:= AllDataW_0;
		FOR KK:= 1 TO SIZEOF(AllDataWPulse) DO 
			Buffer_Rtc[KK]	:= FALSE;
		END_FOR 
	END_IF
END_METHOD

METHOD M_UpdateParameters : BOOL
VAR_INPUT
END_VAR
(*
// Update Parameters
FB_WriteOnChange[1](VarInput := ADR(AllDataParameterWrite.PP_ParamPmax) , VarOut := ADR(A1_PP.ParamPmax), Size:=SIZEOF(A1_PP.ParamPmax) ); 
FB_WriteOnChange[2](VarInput := ADR(AllDataParameterWrite.PP_ParamPmin) , VarOut := ADR(A1_PP.ParamPmin), Size:=SIZEOF(A1_PP.ParamPmin) ); 
FB_WriteOnChange[3](VarInput := ADR(AllDataParameterWrite.PP_ParamQmax) , VarOut := ADR(A1_PP.ParamQmax), Size:=SIZEOF(A1_PP.ParamQmax) ); 
FB_WriteOnChange[4](VarInput := ADR(AllDataParameterWrite.PP_ParamQmin) , VarOut := ADR(A1_PP.ParamQmin), Size:=SIZEOF(A1_PP.ParamQmin) ); 
FB_WriteOnChange[5](VarInput := ADR(AllDataParameterWrite.PP_ParamNominalVoltage) , VarOut := ADR(A1_PP.ParamNominalVoltage), Size:=SIZEOF(A1_PP.ParamNominalVoltage) ); 
FB_WriteOnChange[6](VarInput := ADR(AllDataParameterWrite.PP_ParamNominalFrequency) , VarOut := ADR(A1_PP.ParamNominalFrequency), Size:=SIZEOF(A1_PP.ParamNominalFrequency) ); 
FB_WriteOnChange[7](VarInput := ADR(AllDataParameterWrite.PP_ParamQmaxPbelow20) , VarOut := ADR(A1_PP.ParamQmaxPbelow20), Size:=SIZEOF(A1_PP.ParamQmaxPbelow20) ); 
FB_WriteOnChange[8](VarInput := ADR(AllDataParameterWrite.PP_ParamTanPhiMax) , VarOut := ADR(A1_PP.ParamTanPhiMax), Size:=SIZEOF(A1_PP.ParamTanPhiMax) ); 
FB_WriteOnChange[9](VarInput := ADR(AllDataParameterWrite.PP_ParamTanPhiMin) , VarOut := ADR(A1_PP.ParamTanPhiMin), Size:=SIZEOF(A1_PP.ParamTanPhiMin) ); 
FB_WriteOnChange[10](VarInput := ADR(AllDataParameterWrite.PP_ParamLocalMode) , VarOut := ADR(A1_PP.ParamLocalMode), Size:=SIZEOF(A1_PP.ParamLocalMode) ); 
FB_WriteOnChange[11](VarInput := ADR(AllDataParameterWrite.PP_ParamQcontrol) , VarOut := ADR(A1_PP.ParamQcontrol), Size:=SIZEOF(A1_PP.ParamQcontrol) ); 
FB_WriteOnChange[12](VarInput := ADR(AllDataParameterWrite.PP_ParamTanPhiCtrl) , VarOut := ADR(A1_PP.ParamTanPhiCtrl), Size:=SIZEOF(A1_PP.ParamTanPhiCtrl) ); 
FB_WriteOnChange[13](VarInput := ADR(AllDataParameterWrite.PP_Param_SetptTanPhi) , VarOut := ADR(A1_PP.Param_SetptTanPhi), Size:=SIZEOF(A1_PP.Param_SetptTanPhi) ); 
FB_WriteOnChange[14](VarInput := ADR(AllDataParameterWrite.PP_ParamPoffset_OL) , VarOut := ADR(A1_PP.ParamPoffset_OL), Size:=SIZEOF(A1_PP.ParamPoffset_OL) ); 
FB_WriteOnChange[15](VarInput := ADR(AllDataParameterWrite.PP_ParamQoffset_OL) , VarOut := ADR(A1_PP.ParamQoffset_OL), Size:=SIZEOF(A1_PP.ParamQoffset_OL) ); 
FB_WriteOnChange[16](VarInput := ADR(AllDataParameterWrite.PP_ParamPIDP_K) , VarOut := ADR(A1_PP.ParamPIDP_K), Size:=SIZEOF(A1_PP.ParamPIDP_K) ); 
FB_WriteOnChange[17](VarInput := ADR(AllDataParameterWrite.PP_ParamPidP_I) , VarOut := ADR(A1_PP.ParamPidP_I), Size:=SIZEOF(A1_PP.ParamPidP_I) ); 
FB_WriteOnChange[18](VarInput := ADR(AllDataParameterWrite.PP_ParamPidP_D) , VarOut := ADR(A1_PP.ParamPidP_D), Size:=SIZEOF(A1_PP.ParamPidP_D) ); 
FB_WriteOnChange[19](VarInput := ADR(AllDataParameterWrite.PP_ParamPIDQ_K) , VarOut := ADR(A1_PP.ParamPIDQ_K), Size:=SIZEOF(A1_PP.ParamPIDQ_K) ); 
FB_WriteOnChange[20](VarInput := ADR(AllDataParameterWrite.PP_ParamPidQ_I) , VarOut := ADR(A1_PP.ParamPidQ_I), Size:=SIZEOF(A1_PP.ParamPidQ_I) ); 
FB_WriteOnChange[21](VarInput := ADR(AllDataParameterWrite.PP_ParamPidQ_D) , VarOut := ADR(A1_PP.ParamPidQ_D), Size:=SIZEOF(A1_PP.ParamPidQ_D) ); 
FB_WriteOnChange[22](VarInput := ADR(AllDataParameterWrite.PP_ParamPIDQMin) , VarOut := ADR(A1_PP.ParamPIDQMin), Size:=SIZEOF(A1_PP.ParamPIDQMin) ); 
FB_WriteOnChange[23](VarInput := ADR(AllDataParameterWrite.PP_ParamPIDQMax) , VarOut := ADR(A1_PP.ParamPIDQMax), Size:=SIZEOF(A1_PP.ParamPIDQMax) ); 
FB_WriteOnChange[24](VarInput := ADR(AllDataParameterWrite.PP_ParamQfUQmin) , VarOut := ADR(A1_PP.ParamQfUQmin), Size:=SIZEOF(A1_PP.ParamQfUQmin) ); 
FB_WriteOnChange[25](VarInput := ADR(AllDataParameterWrite.PP_ParamQfUQmax) , VarOut := ADR(A1_PP.ParamQfUQmax), Size:=SIZEOF(A1_PP.ParamQfUQmax) ); 
FB_WriteOnChange[26](VarInput := ADR(AllDataParameterWrite.PP_ParamQfUUHigh) , VarOut := ADR(A1_PP.ParamQfUUHigh), Size:=SIZEOF(A1_PP.ParamQfUUHigh) ); 
FB_WriteOnChange[27](VarInput := ADR(AllDataParameterWrite.PP_ParamQfUDdBandHigh) , VarOut := ADR(A1_PP.ParamQfUDdBandHigh), Size:=SIZEOF(A1_PP.ParamQfUDdBandHigh) ); 
FB_WriteOnChange[28](VarInput := ADR(AllDataParameterWrite.PP_ParamQfUDdBandLow) , VarOut := ADR(A1_PP.ParamQfUDdBandLow), Size:=SIZEOF(A1_PP.ParamQfUDdBandLow) ); 
FB_WriteOnChange[29](VarInput := ADR(AllDataParameterWrite.PP_ParamQfUULow) , VarOut := ADR(A1_PP.ParamQfUULow), Size:=SIZEOF(A1_PP.ParamQfUULow) ); 
FB_WriteOnChange[30](VarInput := ADR(AllDataParameterWrite.PP_ParamNofeedingTime) , VarOut := ADR(A1_PP.ParamNofeedingTime), Size:=SIZEOF(A1_PP.ParamNofeedingTime) ); 
FB_WriteOnChange[31](VarInput := ADR(AllDataParameterWrite.PP_ParamNofeedingWarningTime) , VarOut := ADR(A1_PP.ParamNofeedingWarningTime), Size:=SIZEOF(A1_PP.ParamNofeedingWarningTime) ); 
FB_WriteOnChange[32](VarInput := ADR(AllDataParameterWrite.PP_ParamNofeedingAlarmTime) , VarOut := ADR(A1_PP.ParamNofeedingAlarmTime), Size:=SIZEOF(A1_PP.ParamNofeedingAlarmTime) ); 
FB_WriteOnChange[33](VarInput := ADR(AllDataParameterWrite.PP_ParamDiscoAlarmTime) , VarOut := ADR(A1_PP.ParamDiscoAlarmTime), Size:=SIZEOF(A1_PP.ParamDiscoAlarmTime) ); 
FB_WriteOnChange[34](VarInput := ADR(AllDataParameterWrite.PP_ParamForcedStayConnect) , VarOut := ADR(A1_PP.ParamForcedStayConnect), Size:=SIZEOF(A1_PP.ParamForcedStayConnect) ); 
FB_WriteOnChange[35](VarInput := ADR(AllDataParameterWrite.PP_ParamMinimalDiskSpace) , VarOut := ADR(A1_PP.ParamMinimalDiskSpace), Size:=SIZEOF(A1_PP.ParamMinimalDiskSpace) ); 
FB_WriteOnChange[36](VarInput := ADR(AllDataParameterWrite.PP_ParamCodeVersion) , VarOut := ADR(A1_PP.ParamCodeVersion), Size:=SIZEOF(A1_PP.ParamCodeVersion) ); 
FB_WriteOnChange[37](VarInput := ADR(AllDataParameterWrite.PP_ParamNbCoupler) , VarOut := ADR(A1_PP.ParamNbCoupler), Size:=SIZEOF(A1_PP.ParamNbCoupler) ); 
FB_WriteOnChange[38](VarInput := ADR(AllDataParameterWrite.PTR_1_ParamPTRVersion) , VarOut := ADR(AX_PTR[1].ParamPTRVersion), Size:=SIZEOF(AX_PTR[1].ParamPTRVersion) ); 
FB_WriteOnChange[39](VarInput := ADR(AllDataParameterWrite.PTR_2_ParamPTRVersion) , VarOut := ADR(AX_PTR[2].ParamPTRVersion), Size:=SIZEOF(AX_PTR[2].ParamPTRVersion) ); 
FB_WriteOnChange[40](VarInput := ADR(AllDataParameterWrite.PTR_3_ParamPTRVersion) , VarOut := ADR(AX_PTR[3].ParamPTRVersion), Size:=SIZEOF(AX_PTR[3].ParamPTRVersion) ); 
FB_WriteOnChange[41](VarInput := ADR(AllDataParameterWrite.PTR_4_ParamPTRVersion) , VarOut := ADR(AX_PTR[4].ParamPTRVersion), Size:=SIZEOF(AX_PTR[4].ParamPTRVersion) ); 
FB_WriteOnChange[42](VarInput := ADR(AllDataParameterWrite.PTR_1_ParamTimeOutStart) , VarOut := ADR(AX_PTR[1].ParamTimeOutStart), Size:=SIZEOF(AX_PTR[1].ParamTimeOutStart) ); 
FB_WriteOnChange[43](VarInput := ADR(AllDataParameterWrite.PTR_2_ParamTimeOutStart) , VarOut := ADR(AX_PTR[2].ParamTimeOutStart), Size:=SIZEOF(AX_PTR[2].ParamTimeOutStart) ); 
FB_WriteOnChange[44](VarInput := ADR(AllDataParameterWrite.PTR_3_ParamTimeOutStart) , VarOut := ADR(AX_PTR[3].ParamTimeOutStart), Size:=SIZEOF(AX_PTR[3].ParamTimeOutStart) ); 
FB_WriteOnChange[45](VarInput := ADR(AllDataParameterWrite.PTR_4_ParamTimeOutStart) , VarOut := ADR(AX_PTR[4].ParamTimeOutStart), Size:=SIZEOF(AX_PTR[4].ParamTimeOutStart) ); 
FB_WriteOnChange[46](VarInput := ADR(AllDataParameterWrite.PTR_1_ParamTimeOutStop) , VarOut := ADR(AX_PTR[1].ParamTimeOutStop), Size:=SIZEOF(AX_PTR[1].ParamTimeOutStop) ); 
FB_WriteOnChange[47](VarInput := ADR(AllDataParameterWrite.PTR_2_ParamTimeOutStop) , VarOut := ADR(AX_PTR[2].ParamTimeOutStop), Size:=SIZEOF(AX_PTR[2].ParamTimeOutStop) ); 
FB_WriteOnChange[48](VarInput := ADR(AllDataParameterWrite.PTR_3_ParamTimeOutStop) , VarOut := ADR(AX_PTR[3].ParamTimeOutStop), Size:=SIZEOF(AX_PTR[3].ParamTimeOutStop) ); 
FB_WriteOnChange[49](VarInput := ADR(AllDataParameterWrite.PTR_4_ParamTimeOutStop) , VarOut := ADR(AX_PTR[4].ParamTimeOutStop), Size:=SIZEOF(AX_PTR[4].ParamTimeOutStop) ); 
FB_WriteOnChange[50](VarInput := ADR(AllDataParameterWrite.PTR_1_ParamTimeOutDisconnect) , VarOut := ADR(AX_PTR[1].ParamTimeOutDisconnect), Size:=SIZEOF(AX_PTR[1].ParamTimeOutDisconnect) ); 
FB_WriteOnChange[51](VarInput := ADR(AllDataParameterWrite.PTR_2_ParamTimeOutDisconnect) , VarOut := ADR(AX_PTR[2].ParamTimeOutDisconnect), Size:=SIZEOF(AX_PTR[2].ParamTimeOutDisconnect) ); 
FB_WriteOnChange[52](VarInput := ADR(AllDataParameterWrite.PTR_3_ParamTimeOutDisconnect) , VarOut := ADR(AX_PTR[3].ParamTimeOutDisconnect), Size:=SIZEOF(AX_PTR[3].ParamTimeOutDisconnect) ); 
FB_WriteOnChange[53](VarInput := ADR(AllDataParameterWrite.PTR_4_ParamTimeOutDisconnect) , VarOut := ADR(AX_PTR[4].ParamTimeOutDisconnect), Size:=SIZEOF(AX_PTR[4].ParamTimeOutDisconnect) ); 
FB_WriteOnChange[54](VarInput := ADR(AllDataParameterWrite.PTR_1_ParamTempoComAlarm) , VarOut := ADR(AX_PTR[1].ParamTempoComAlarm), Size:=SIZEOF(AX_PTR[1].ParamTempoComAlarm) ); 
FB_WriteOnChange[55](VarInput := ADR(AllDataParameterWrite.PTR_2_ParamTempoComAlarm) , VarOut := ADR(AX_PTR[2].ParamTempoComAlarm), Size:=SIZEOF(AX_PTR[2].ParamTempoComAlarm) ); 
FB_WriteOnChange[56](VarInput := ADR(AllDataParameterWrite.PTR_3_ParamTempoComAlarm) , VarOut := ADR(AX_PTR[3].ParamTempoComAlarm), Size:=SIZEOF(AX_PTR[3].ParamTempoComAlarm) ); 
FB_WriteOnChange[57](VarInput := ADR(AllDataParameterWrite.PTR_4_ParamTempoComAlarm) , VarOut := ADR(AX_PTR[4].ParamTempoComAlarm), Size:=SIZEOF(AX_PTR[4].ParamTempoComAlarm) ); 
FB_WriteOnChange[58](VarInput := ADR(AllDataParameterWrite.PTR_1_ParamTempoStartInv) , VarOut := ADR(AX_PTR[1].ParamTempoStartInv), Size:=SIZEOF(AX_PTR[1].ParamTempoStartInv) ); 
FB_WriteOnChange[59](VarInput := ADR(AllDataParameterWrite.PTR_2_ParamTempoStartInv) , VarOut := ADR(AX_PTR[2].ParamTempoStartInv), Size:=SIZEOF(AX_PTR[2].ParamTempoStartInv) ); 
FB_WriteOnChange[60](VarInput := ADR(AllDataParameterWrite.PTR_3_ParamTempoStartInv) , VarOut := ADR(AX_PTR[3].ParamTempoStartInv), Size:=SIZEOF(AX_PTR[3].ParamTempoStartInv) ); 
FB_WriteOnChange[61](VarInput := ADR(AllDataParameterWrite.PTR_4_ParamTempoStartInv) , VarOut := ADR(AX_PTR[4].ParamTempoStartInv), Size:=SIZEOF(AX_PTR[4].ParamTempoStartInv) ); 
FB_WriteOnChange[62](VarInput := ADR(AllDataParameterWrite.PTR_1_ParamTempoStopInv) , VarOut := ADR(AX_PTR[1].ParamTempoStopInv), Size:=SIZEOF(AX_PTR[1].ParamTempoStopInv) ); 
FB_WriteOnChange[63](VarInput := ADR(AllDataParameterWrite.PTR_2_ParamTempoStopInv) , VarOut := ADR(AX_PTR[2].ParamTempoStopInv), Size:=SIZEOF(AX_PTR[2].ParamTempoStopInv) ); 
FB_WriteOnChange[64](VarInput := ADR(AllDataParameterWrite.PTR_3_ParamTempoStopInv) , VarOut := ADR(AX_PTR[3].ParamTempoStopInv), Size:=SIZEOF(AX_PTR[3].ParamTempoStopInv) ); 
FB_WriteOnChange[65](VarInput := ADR(AllDataParameterWrite.PTR_4_ParamTempoStopInv) , VarOut := ADR(AX_PTR[4].ParamTempoStopInv), Size:=SIZEOF(AX_PTR[4].ParamTempoStopInv) ); 
FB_WriteOnChange[66](VarInput := ADR(AllDataParameterWrite.PTR_1_ParamPTRNum) , VarOut := ADR(AX_PTR[1].ParamPTRNum), Size:=SIZEOF(AX_PTR[1].ParamPTRNum) ); 
FB_WriteOnChange[67](VarInput := ADR(AllDataParameterWrite.PTR_2_ParamPTRNum) , VarOut := ADR(AX_PTR[2].ParamPTRNum), Size:=SIZEOF(AX_PTR[2].ParamPTRNum) ); 
FB_WriteOnChange[68](VarInput := ADR(AllDataParameterWrite.PTR_3_ParamPTRNum) , VarOut := ADR(AX_PTR[3].ParamPTRNum), Size:=SIZEOF(AX_PTR[3].ParamPTRNum) ); 
FB_WriteOnChange[69](VarInput := ADR(AllDataParameterWrite.PTR_4_ParamPTRNum) , VarOut := ADR(AX_PTR[4].ParamPTRNum), Size:=SIZEOF(AX_PTR[4].ParamPTRNum) ); 
FB_WriteOnChange[70](VarInput := ADR(AllDataParameterWrite.PTR_1_ParamNbINV) , VarOut := ADR(AX_PTR[1].ParamNbINV), Size:=SIZEOF(AX_PTR[1].ParamNbINV) ); 
FB_WriteOnChange[71](VarInput := ADR(AllDataParameterWrite.PTR_2_ParamNbINV) , VarOut := ADR(AX_PTR[2].ParamNbINV), Size:=SIZEOF(AX_PTR[2].ParamNbINV) ); 
FB_WriteOnChange[72](VarInput := ADR(AllDataParameterWrite.PTR_3_ParamNbINV) , VarOut := ADR(AX_PTR[3].ParamNbINV), Size:=SIZEOF(AX_PTR[3].ParamNbINV) ); 
FB_WriteOnChange[73](VarInput := ADR(AllDataParameterWrite.PTR_4_ParamNbINV) , VarOut := ADR(AX_PTR[4].ParamNbINV), Size:=SIZEOF(AX_PTR[4].ParamNbINV) ); 
FB_WriteOnChange[74](VarInput := ADR(AllDataParameterWrite.SUBMV_ParamTempoPoste) , VarOut := ADR(A1_SUBMV.ParamTempoPoste), Size:=SIZEOF(A1_SUBMV.ParamTempoPoste) ); 
FB_WriteOnChange[75](VarInput := ADR(AllDataParameterWrite.SUBMV_ParamTempoUnknowFault) , VarOut := ADR(A1_SUBMV.ParamTempoUnknowFault), Size:=SIZEOF(A1_SUBMV.ParamTempoUnknowFault) ); 
FB_WriteOnChange[76](VarInput := ADR(AllDataParameterWrite.SUBMV_ParamTempoSepamCloseAfterGte) , VarOut := ADR(A1_SUBMV.ParamTempoSepamCloseAfterGte), Size:=SIZEOF(A1_SUBMV.ParamTempoSepamCloseAfterGte) ); 
FB_WriteOnChange[77](VarInput := ADR(AllDataParameterWrite.SUBMV_ParamAutoCloseMainMVCBEnabled) , VarOut := ADR(A1_SUBMV.ParamAutoCloseMainMVCBEnabled), Size:=SIZEOF(A1_SUBMV.ParamAutoCloseMainMVCBEnabled) ); 
FB_WriteOnChange[78](VarInput := ADR(AllDataParameterWrite.SUBMV_ParamSUB_MVVersion) , VarOut := ADR(A1_SUBMV.ParamSUB_MVVersion), Size:=SIZEOF(A1_SUBMV.ParamSUB_MVVersion) ); 
FB_WriteOnChange[79](VarInput := ADR(AllDataParameterWrite.SUBMV_ParamTimeOutConnect) , VarOut := ADR(A1_SUBMV.ParamTimeOutConnect), Size:=SIZEOF(A1_SUBMV.ParamTimeOutConnect) ); 
FB_WriteOnChange[80](VarInput := ADR(AllDataParameterWrite.SUBMV_ParamTimeOutDisconnect) , VarOut := ADR(A1_SUBMV.ParamTimeOutDisconnect), Size:=SIZEOF(A1_SUBMV.ParamTimeOutDisconnect) ); 
FB_WriteOnChange[81](VarInput := ADR(AllDataParameterWrite.SUBMV_ParamTempoComAlarm) , VarOut := ADR(A1_SUBMV.ParamTempoComAlarm), Size:=SIZEOF(A1_SUBMV.ParamTempoComAlarm) ); 
FB_WriteOnChange[82](VarInput := ADR(AllDataParameterWrite.SUBMV_ParamPmax) , VarOut := ADR(A1_SUBMV.ParamPmax), Size:=SIZEOF(A1_SUBMV.ParamPmax) ); 
FB_WriteOnChange[83](VarInput := ADR(AllDataParameterWrite.SUBMV_ParamPmin) , VarOut := ADR(A1_SUBMV.ParamPmin), Size:=SIZEOF(A1_SUBMV.ParamPmin) ); 
FB_WriteOnChange[84](VarInput := ADR(AllDataParameterWrite.WS_ParamDurationIntegerGTI) , VarOut := ADR(A1_WS.ParamDurationIntegerGTI), Size:=SIZEOF(A1_WS.ParamDurationIntegerGTI) ); 
*)
END_METHOD

METHOD M_Wago
VAR_INPUT
END_VAR
(*
OpcUaServer_1:=  OpcUa.AllDataR.PP.MesU ; 
OpcUaServer_2:=  OpcUa.AllDataR.PP.MesFreq ; 
OpcUaServer_3:=  OpcUa.AllDataR.PP.OUT_SetptP ; 
OpcUaServer_4:=  OpcUa.AllDataR.PP.OUT_SetptQ ; 
OpcUaServer_5:=  OpcUa.AllDataR.PTR[1].MesDataExd.MesData.MesP ; 
OpcUaServer_6:=  OpcUa.AllDataR.PTR[1].MesDataExd.MesData.MesQ ; 
OpcUaServer_7:=  OpcUa.AllDataR.PTR[1].MesDataExd.MesData.MesI ; 
OpcUaServer_8:=  OpcUa.AllDataR.SUBMV.MesDataExd.MesData.MesU ; 
OpcUaServer_9:=  OpcUa.AllDataR.SUBMV.MesDataExd.MesData.MesFreq ; 
OpcUaServer_10:=  OpcUa.AllDataR.WS.MesGTI ; 
OpcUaServer_11:=  OpcUa.AllDataR.WS.MesGHI ; 
OpcUaServer_12:=  OpcUa.AllDataR.PTR[1].AX_INV[1].MesDataExd.MesData.MesP ; 
OpcUaServer_13:=  OpcUa.AllDataR.PTR[1].AX_INV[1].MesDataExd.MesData.MesQ ; 
OpcUaServer_14:=  OpcUa.AllDataR.PTR[1].AX_INV[1].MesDataExd.MesData.MesPdc ; 
OpcUaServer_15:=  OpcUa.AllDataR.PTR[1].AX_INV[1].MesDataExd.MesData.MesUdc ; 
OpcUaServer_16:=  OpcUa.AllDataR.PTR[1].AX_INV[1].MesDataExd.MesData.MesU ; 
OpcUaServer_17:=  OpcUa.AllDataR.PTR[1].AX_INV[1].MesDataExd.MesData.MesI ; 
OpcUaServer_18:=  OpcUa.AllDataR.PTR[1].AX_INV[1].MesDataExd.MesData.MesFreq ; 
OpcUaServer_19:=  OpcUa.AllDataR.PTR[1].AX_INV[1].MesDataExd.MesData.OUT_SetptP ; 
OpcUaServer_20:=  OpcUa.AllDataR.PTR[1].AX_INV[1].MesDataExd.MesData.OUT_SetptQ ; 
OpcUaServer_21:=  OpcUa.AllDataR.SUBMV.GRID.MesDataExd.MesData.OUT_SetptP ; 
OpcUaServer_22:=  OpcUa.AllDataR.SUBMV.GRID.MesDataExd.MesData.OUT_SetptQ ; 
OpcUaServer_23:=  OpcUa.AllDataR.SUBMV.ProtectRelay_Freq.MesI  ; 
OpcUaServer_24:=  OpcUa.AllDataR.SUBMV.ProtectRelay_Freq.MesFreq ; 
OpcUaServer_25:=  OpcUa.AllDataR.SUBMV.PM.MesFreq ; 
OpcUaServer_26:=  OpcUa.AllDataR.SUBMV.PM.MesP ; 
OpcUaServer_27:=  OpcUa.AllDataR.SUBMV.PM.MesQ ; 
OpcUaServer_28:=  OpcUa.AllDataR.SUBMV.PM.MesI ; 
OpcUaServer_29:=  OpcUa.AllDataR.SUBMV.PM.MesU ; 
OpcUaServer_30:=  OpcUa.AllDataR.SUBMV.ProtectRelay_Freq.MesI ; 
OpcUaServer_31:=  OpcUa.AllDataR.SUBMV.ProtectRelay_Freq.MesFreq ; 
OpcUaServer_32:=  OpcUa.AllDataR.WS.Pyran_GHI_1.Value ; 
OpcUaServer_33:=  OpcUa.AllDataR.WS.Pyran_GHI_2.Value ; 
OpcUaServer_34:=  OpcUa.AllDataR.WS.Pyran_GTI_1.Value ; 
OpcUaServer_35:=  OpcUa.AllDataR.WS.Pyran_GTI_2.Value ; 
OpcUaServer_36:=  OpcUa.AllDataR.WS.TempSensor_Ext.Value ; 
OpcUaServer_37:=  OpcUa.AllDataR.WS.windDir.Value ; 
OpcUaServer_38:=  OpcUa.AllDataR.WS.WindSp.Value ; 
OpcUaServer_39:=  OpcUa.AllDataR.WS.Rain.AvgmmHour ; 
OpcUaServer_40:=  OpcUa.AllDataR.WS.Rain.AvgmmDay ; 
OpcUaServer_41:=  OpcUa.AllDataR.WS.Rain.AvgmmMonth ; 
OpcUaServer_42:=  OpcUa.AllDataR.WS.TempSensor_Panel_PTR1.Value ; 
OpcUaServer_43:=  OpcUa.AllDataR.WS.TempSensor_Panel_PTR2.Value ; 
*)
END_METHOD

END_PROGRAM

// ---- 00_FunctionsBlocks/Common/BoolManagement/FB_TapVariable.TcPOU
FUNCTION_BLOCK FB_TapVariable
////////////////// 
// TAp a variable when input is active and reset after 
//////////////////	

VAR_IN_OUT
	TapOut			: BOOL;		// Output VTap Variable
	
END_VAR

VAR_INPUT
	TapTrigger		: BOOL;		// Input Trigger
	
END_VAR

VAR
	F_TRIG_Trigger	: F_TRIG;	// Trigger detection 
	R_TRIG_Trigger	: R_TRIG;	// Trigger detection 		
	
	
END_VAR

R_TRIG_Trigger(CLK:= TapTrigger);
F_TRIG_Trigger(CLK:= TapTrigger);

IF R_TRIG_Trigger.Q THEN
	TapOut			:=TRUE;
	
ELSIF F_TRIG_Trigger.Q  THEN 
	TapOut			:=FALSE ;
			
END_IF

END_FUNCTION_BLOCK

// ---- 00_FunctionsBlocks/Beckhoff/AlarmManagement/SMS_Server.TcPOU
PROGRAM SMS_Server
VAR PERSISTENT
	AX_Numtel						: ARRAY[1..CstNbUser] OF STRING(26) ;	//Contient tous les numéros des utilisateurs
	AX_Subscribed					: ARRAY[1..CstNbUser] OF BOOL ;			//Contient tous les états d'abonnements des utilisateurs aux SMS
	AX_NomUtili						: ARRAY[1..CstNbUser] OF STRING(50);	//Contient tous les noms des utilisateurs
	AX_User_LVL						: ARRAY[1..CstNbUser] OF WORD;			//Contient tous les niveau d'adhésion des utilisateurs.
END_VAR

VAR_INPUT
	IN_DataSetFifo_ReadSMS			: FB_SMSDatasetFifo_Read; //Buffer automate des sms récuperer depuis modem Gsm
	IN_DataSetFifo_SendSMS			: FB_SMSDatasetFifo_Send; //Buffer automate des sms récuperer depuis modem Gsm	
	IN_AX_Journal					: ARRAY [0..CstNbAlarmCode] OF ARRAY[0..15] OF ST_ValuesAlarms; //Journal d'envoi, contient destinataire et message, et gestion de l'envois ou pas du sms
	IN_Reset_OPC					: BOOL;
	IN_ChangePhoneMailInfos_OPC			: BOOL;
	IN_Reset_SmsServer				: BOOL;
	IN_CmdReset_L					: BOOL;
	IN_CmdDeleteAllSms			: BOOL;
	
	
		MesData			: ServerSMS;
	
END_VAR

VAR
	fbSerialLineControl		: SerialLineControl;
	stTxBufferPC			: ComBuffer;
	stRxBufferPC			: ComBuffer;
	fbReadSMS				: FB_ReadSMS;
	fbSendSMS				: FB_SendSMS;
	fbDeleteSMS				: FB_DeleteSMS;
	fbDeleteAllSMS			: FB_DeleteAllSMS;
	Fblogin 				: FB_Login;
	
	//READ VARIABLE 
	bStartRead				: BOOL; //Gestion du front montant FB ReadSMS
	ReadSMS_bBusy			: BOOL;
	ReadSMS_bError			: BOOL;
	ReadSMS_nErrorID		: UINT;
	
	LoginSMS_bError			: BOOL;
	LoginSMS_bBusy		    : BOOL;
	IndexReadMessage		: USINT:=1; //Index du message a lire
	ReadSMS_MessageText		: STRING(240); // Message brut du SMS recu
	Etape_Read 		 		: SINT:=0; // Etape du Case de M_Fill_Buffer_Read
	Message_Tous_lu 		: BOOL;  // Si tous les message du buffer READ sont lu : True sinon False
	
	//DELETE VARIABLE
	bStartDelete			: BOOL; //Gestion du front montant FB DeleteSms
	DeletedSMS_bBusy		: BOOL;
	DeletedSMS_Error		: BOOL;
	DeletedSMS_nErrorID		: UINT;
	
	IndexDeleteMessage 		: USINT:=1; //Index du message a supprimer
	
	//SEND VARIABLE
	bStartSend				: BOOL;
	Message_Send			: STRING(160);
	MesTimeStamp			: STRING(17);
	SendSMS_bBusy			: BOOL;
	SendSMS_bError			: BOOL;
	Etape_Send				: SINT;
	CPT						: SINT:=1;
	Num_Tel					: STRING(30);

	//INIT VARIABLE
	bStartlogin             : BOOL:=TRUE; //Gestion du front montant FB login
	bInit					: BOOL;
	
	//Variables de All Delete
	DeletedAllSMS_bBusy		: BOOL;
	DeletedAllSMS_Error		: BOOL;
	DeletedAllSMS_nErrorID	: UINT;
	G7_DelAll				: SINT;

	Bstart_delete_all		: BOOL;    
	
	//M_G7_SMS
	CPT_Message				: CTU;
	


	//TABLEAU
	AX_MesAlarmCode_Bool	: ARRAY [1..CstNbAlarmCode] OF ARRAY[1..15] OF BOOL; //Tableau de tous les alarmesCode en Bool
	AX_Alarm_State			: ARRAY [1..CstNbAlarmCode] OF ARRAY[1..15] OF BOOL; //Tableau de Bool avec toutes les nouveaux bit modifiés
	fbXorWord				: FB_XorWord; //Compare 2 Word et retourne les bit modifié
	Extract_Num_Mes			: FB_Extract_Num_Mes; //Extraction des infos: Message,Numero de tel

	// M_Evaluate

	CalNbrUtiliActive    : INT := 10;
	//AlarmCode
	RS_LoginSMS_bError		: RS;
	RS_SendSMS_bError       : RS;
	RS_ReadSMS_bError       : RS;
	RS_DeletedSMS_Error     : RS;
    RS_DeletedAllSMS_Error  : RS;

	AX_Cmd_SMS				: ARRAY[1..CstNbCMD] OF STRING(26):=['Infos','Reboot_ADSL','P_Onduleur','Stop_SMS','Start_SMS','Toggle subscription','Ip Publique','Active Alarms','Help','Test SMS','ForcedStayConnect','Restart Telegraf','Restart PLC','Auto Couplage','Disconnect', 'VPN Connect', 'VPN Disconnect', 'Reboot_IPC']; //Contient toutes les commandes possibles

	Serial_Use				: BOOL:=TRUE;
	ReadAct					: BOOL:=FALSE;
	LoginOK                 : BOOL:=TRUE;
	Reset					: BOOL;
	
	//OPC
	RS_OPC					: RS;
	RS_Deletteall			: RS;
	RS_Reset				: RS;
	Trig_OPC				: R_TRIG;
	Trig_OpcDelAll			: R_TRIG;
	Trig_OpcReset			: R_TRIG;

	
	
END_VAR

IF NOT bInit THEN
	M_Init();
ELSE
	
	// READ OPC Data .
	M_OPC();

	//SERIALLINEMODE_EL6_22B	
	fbSerialLineControl(Mode:= SERIALLINEMODE_PC_COM_PORT ,
		pComIn:= ADR(stPCComInData),
		pComOut:= ADR(stPCComOutData),
		SizeComIn:= UINT_TO_INT( SIZEOF(stPCComInData)),
		TxBuffer:= stTxBufferPC,
		RxBuffer:= stRxBufferPC,
		Error=> ,
		ErrorID=> );
		
	Fblogin(bStart:=bStartlogin ,					// etrangement le login fonctionne puis fait une erreur , puis refonctionne etc . relance du login sur read error je pense qui entraine une tentative de login qui foire. 	
			stTxBuffer:=stTxBufferPC,	
			stRxBuffer:=stRxBufferPC,
			bBusy =>LoginSMS_bBusy,
			bError=>LoginSMS_bError
			);		
		
	fbSendSMS(bStart:= bStartSend,
		sPhoneNumber:= Num_Tel,
		bReset := IN_Reset_OPC ,
		sSMSText:= Message_Send,
		stTxBuffer:=stTxBufferPC ,
		stRxBuffer:=stRxBufferPC,
		bBusy=>SendSMS_bBusy,
		bError=>SendSMS_bError);
	
	fbReadSMS(bStart:= bStartRead,
		nIndex:= IndexReadMessage,
		stTxBuffer:=stTxBufferPC ,
		stRxBuffer:=stRxBufferPC ,
		bBusy=> ReadSMS_bBusy,
		bError=> ReadSMS_bError,
		nErrorID=> ReadSMS_nErrorID
		);
	
	
	fbDeleteSMS
	(
		bStart:= bStartDelete,
		nIndex:= IndexDeleteMessage,
		stTxBuffer:=stTxBufferPC,
		stRxBuffer:=stRxBufferPC,
		bBusy=> DeletedSMS_bBusy,
		bError=> DeletedSMS_Error,
		nErrorID=> DeletedSMS_nErrorID
	);
	
	fbDeleteAllSMS
	(
		bStart:= Bstart_delete_all,
		stTxBuffer:=stTxBufferPC,
		stRxBuffer:=stRxBufferPC,
		bBusy=> DeletedAllSMS_bBusy,
		bError=> DeletedAllSMS_Error,
		nErrorID=> DeletedAllSMS_nErrorID
	);	

	M_DeleteAll();
	M_Fill_Buffer_Read(); //Lecture de tous les messages recu

	M_AlarmManager();
	M_Evaluate();		// Update serveur info
	M_Send(); // Envois de tous les messages (Alarm ou réponce aux sms de cmd)

	M_Cmd_Execute(); // Verification des messages recu
	
	IF Reset OR IN_Reset_OPC  THEN
		M_Reset();
	END_IF
	
	IF NOT LoginSMS_bBusy AND NOT LoginSMS_bError AND LoginOK THEN
		BstartLogin := FALSE;
		Serial_Use:=FALSE;
		LoginOK:=FALSE;
	END_IF
	
	
END_IF

METHOD M_AlarmManager
VAR
	ii:SINT;
	jj:INT;
	KK:INT;
	FB_AlarmCodeManager			: FB_AlarmCodeManager ;
END_VAR
RS_LoginSMS_bError(SET:=LoginSMS_bError,RESET1:=	IN_CmdReset_L OR IN_Reset_OPC); 		
RS_SendSMS_bError(SET:=SendSMS_bError,RESET1:=  	IN_CmdReset_L OR IN_Reset_OPC); 		
RS_ReadSMS_bError(SET:=ReadSMS_bError,RESET1:=  	IN_CmdReset_L OR IN_Reset_OPC); 		
RS_DeletedSMS_Error(SET:=DeletedSMS_Error,RESET1:=	IN_CmdReset_L OR IN_Reset_OPC); 		
RS_DeletedAllSMS_Error(SET:=DeletedAllSMS_Error,RESET1:=IN_CmdReset_L OR IN_Reset_OPC); 	

// ALARM CODE //
	FB_AlarmCodeManager(
		bAlarm1			:= RS_LoginSMS_bErrOR.Q1		  ,			// Login SMS Error
		bAlarm2			:= RS_SendSMS_bErrOR.Q1		   ,			// Send SMS Error
		bAlarm3			:= RS_ReadSMS_bErrOR.Q1		   ,			// Read SMS Error 
		bAlarm4			:= RS_DeletedSMS_ErrOR.Q1		 ,			// Delete SMS Error 
		bAlarm5			:= RS_DeletedAllSMS_ErrOR.Q1	,			// Delete All Sms Error
		bAlarm6			:= IN_DataSetFifo_ReadSMS.bOverwrite,		// Read Fifo overflow
		bAlarm7			:= IN_DataSetFifo_SendSMS.bOverwrite,       // Send Fifo overflow
		bAlarm8			:= FALSE,                                   //
		bAlarm9			:= FALSE,                                   //
		bAlarm10		:= FALSE,                                   //
		bAlarm11		:= FALSE,									//
		bAlarm12		:= FALSE,                                   //
		bAlarm13		:= FALSE,                                   //
		bAlarm14		:= FALSE,                                   //
		bAlarm15		:= FALSE,                                   //
		wAlarmCode		=>MesData.MesAlarmCode);
END_METHOD

METHOD M_Cmd_Execute
VAR_INPUT
END_VAR

VAR
	i: SINT;
	Num_Valide 		: BOOL;
	Message_Valide 	: BOOL;
	Index_CMD 		: SINT;
END_VAR
IF IN_DataSetFifo_ReadSMS.nCount > 0 THEN
	IN_DataSetFifo_ReadSMS.A_Get(); // Récuperation du FIFO
	FOR i:=1 TO CstNbUser DO // VERIFICATION du numéro de telephone
		IF AX_Numtel[i]=IN_DataSetFifo_ReadSMS.Out.Num THEN
			Num_Valide := TRUE;
			EXIT;
		END_IF
	END_FOR
	IF Num_Valide THEN
		FOR i:=1 TO CstNbCMD DO // VERIFICATION du message
			IF IN_DataSetFifo_ReadSMS.Out.Message=AX_Cmd_SMS[i] THEN
				Message_Valide := TRUE;
				Index_CMD:=i;
				EXIT;
			END_IF
		END_FOR
	END_IF
	
	IF Num_Valide AND Message_Valide THEN
		M_G7_SMS(G7_Etape:=Index_CMD);

	ELSE
		IN_DataSetFifo_ReadSMS.A_Remove(); //IL s'agit d'un spam ou d'un utilisateur non autorisé
	END_IF
	

END_IF
END_METHOD

METHOD M_DeleteAll


VAR
	
END_VAR
CASE G7_DelAll OF
	
	0: // Entrée
		IF RS_Deletteall.Q1 AND NOT Serial_Use THEN
			Serial_Use 			:= TRUE;
			Bstart_delete_all 	:= TRUE;
			G7_DelAll 			:= 1;
		END_IF
	1: // attente du bb=usy
		Bstart_delete_all 	:= FALSE;
		IF NOT DeletedAllSMS_bBusy OR DeletedAllSMS_Error THEN
			RS_Deletteall(RESET1:= TRUE);
			RS_Deletteall(RESET1:= FALSE);
			Serial_Use 			:= FALSE;
			G7_DelAll 			:= 0;
		END_IF
		
		
END_CASE
END_METHOD

METHOD M_Evaluate
VAR 
	KK: INT;
END_VAR
CalNbrUtiliActive := 0 ;
FOR KK:=1 TO CstNbUser DO 
	IF 	AX_Numtel[KK] <> '' THEN 
		CalNbrUtiliActive := CalNbrUtiliActive+1 ; 
	END_IF
END_FOR



Mesdata.NbrUtiliActive 	:= CalNbrUtiliActive ;
Mesdata.AX_Numtel		:= AX_Numtel			;
Mesdata.AX_Subscribed	:= AX_subscribed	    ;
MesData.AX_NomUtili		:= AX_NomUtili		    ;
MesData.AX_UserLVL		:= AX_User_LVL		    ;
END_METHOD

METHOD M_Fill_Buffer_Read
CASE Etape_Read OF
	0://Initilisation
		IF NOT ReadSMS_bBusy AND NOT Serial_Use AND ReadAct THEN
			Etape_Read:=10;
			ReadSMS_MessageText:='';
			bStartlogin:=TRUE;
			Serial_Use:=TRUE;
		END_IF
	10: //Initialisation MODEM (ECHO OFF)
		//Serial_Use:=TRUE;
		bStartlogin:=FALSE;
		IF NOT LoginSMS_bBusy AND NOT LoginSMS_bError THEN
			Etape_Read:=1;
			BstartRead:=TRUE;	
		ELSIF LoginSMS_bError THEN
			Etape_Read:=0;
			Serial_Use:=FALSE;
		END_IF
	1://Lecture des sms
		//GVL_Rapale.Serial_Use:=TRUE;
		ReadSMS_MessageText:=fbReadSMS.sMessageText;
		BstartRead:=FALSE;	
		IF NOT ReadSMS_bBusy AND NOT ReadSMS_bError THEN	
			Etape_Read:=2;
			Serial_Use:=FALSE;
		ELSIF ReadSMS_bError THEN
			Etape_Read:=0;
			Serial_Use:=FALSE;
			
		END_IF
		
	2://Analyse du sms en Cas d'un message non vide
		IF(ReadSMS_MessageText<>'OK$R$N') AND (ReadSMS_MessageText<>'') THEN
			
			IF (FIND(ReadSMS_MessageText,'REC UNREAD')>0) THEN		//
				Message_Tous_lu := FALSE;
				IndexReadMessage:=IndexReadMessage+1;
				Extract_Num_Mes(InMessage:=ReadSMS_MessageText);
				IN_DataSetFifo_ReadSMS.A_Add( in := Extract_Num_Mes.OutDataEntry);
				Etape_Read:=0;					
			ELSE	// Messages have already been read. 
				Message_Tous_lu := TRUE;
				IndexReadMessage:=IndexReadMessage+1;
				ReadSMS_MessageText:='';
				Etape_Read:=0;
			END_IF
		ELSE
			Etape_Read:=3;
		END_IF
	3://Analyse du sms en cas de message vide
		IF Message_Tous_lu THEN
			Etape_Read:=4;
		ELSE
			IndexReadMessage:=1;
			Etape_Read:=0;
		END_IF
	4://Initialisation du Delete_FB
		IF NOT DeletedSMS_bBusy AND ReadAct THEN //AND NOT GVL_Rapale.Serial_Use THEN
			Etape_Read:=5;
			bStartDelete:=TRUE;
			Serial_Use:=TRUE;
		END_IF
	5://Suppression du buffer GSM
		//GVL_Rapale.Serial_Use:=TRUE;
			bStartDelete:=FALSE;
		IF NOT DeletedSMS_bBusy AND NOT DeletedSMS_Error THEN
			Serial_Use:=FALSE;
			Etape_Read:=6;
		ELSIF DeletedSMS_Error THEN
			//GVL_Rapale.Serial_Use:=FALSE;
			Etape_Read:=4;
			Serial_Use:=FALSE;
		END_IF
	6://Controle suppression
		IF IndexDeleteMessage=IndexReadMessage-1 THEN
			Etape_Read:=0;
			IndexDeleteMessage:=1;
			Message_Tous_lu:=FALSE;
			IndexReadMessage:=IndexReadMessage+1;
			Serial_Use:=FALSE;
		ELSE
			IndexDeleteMessage:=IndexDeleteMessage+1;
			Etape_Read:=4;
		END_IF		
		
END_CASE
END_METHOD

METHOD M_G7_SMS
VAR_INPUT
	G7_Etape :SINT;
END_VAR

VAR
	InStruct 		: ST_ValuesAlarms;
END_VAR
FUN_Alarms.M_G7_SMS(
	DataSetFifo_ReadSMS		:= IN_DataSetFifo_ReadSMS,
    IN_DataSetFifo_SendSMS	:= IN_DataSetFifo_SendSMS,
 	CPT_Message				:= CPT_Message,	
    InStruct 				:= InStruct,
    G7_Etape 				:= G7_Etape,
    AX_Numtel				:= AX_Numtel,
    AX_subscribed			:= AX_subscribed,
    AX_MesAlarmCode_Bool	:= AX_MesAlarmCode_Bool,
    AX_Cmd_SMS		        := AX_Cmd_SMS
);
END_METHOD

METHOD M_Init

//Initialisation BUFFER

	//Buffer pour la lecture des sms
	IN_DataSetFifo_ReadSMS.A_Reset();
	IN_DataSetFifo_ReadSMS.A_Add();
	IN_DataSetFifo_ReadSMS.A_Get();
	IN_DataSetFifo_ReadSMS.A_Remove();
	
	//Buffer pour l'envois des sms
	IN_DataSetFifo_SendSMS.A_Reset();
	IN_DataSetFifo_SendSMS.A_Add();
	IN_DataSetFifo_SendSMS.A_Get();
	IN_DataSetFifo_SendSMS.A_Remove();

//Initialisation du Journal		
bInit := TRUE;
END_METHOD

METHOD M_OPC : BOOL
VAR
	AX_Numtel_Init				: ARRAY[1..CstNbUser] OF STRING(26);
END_VAR
Trig_OPC(CLK := IN_ChangePhoneMailInfos_OPC);
Trig_OpcDelAll(CLK := IN_CmdDeleteAllSms);
Trig_OpcReset(CLK:= IN_Reset_SmsServer);

RS_OPC(SET:= Trig_OPC.Q);
RS_Deletteall(SET:=Trig_OpcDelAll.Q);
RS_Reset(Set:=Trig_OpcReset.Q);

IF (*NOT Serial_Use AND*) RS_OPC.Q1 THEN
	//Numéro de téléphone
	AX_Numtel := OpcUa.AllValueW.AX_NbPhone_OPC;
	//Nom d'utilisateur
	AX_NomUtili	:= OpcUa.AllValueW.AX_NamesUsers_OPC;
	
	// User LVL . 
	AX_User_LVL := OpcUa.AllValueW.AX_UserLVL;

	//Gestion subscription
	AX_Subscribed := OpcUa.AllValueW.AX_SubscribedSms_OPC;

	RS_OPC(RESET1:= TRUE);
	RS_OPC(Reset1 := FALSE);
END_IF

IF RS_Reset.Q1 THEN
	IN_Reset_Opc := TRUE;
END_IF
END_METHOD

METHOD M_Reset : BOOL
VAR_INPUT
END_VAR
IN_DataSetFifo_SendSMS.A_Reset();

bStartRead 		:= FALSE;
bStartSend 		:= FALSE;
bStartDelete 	:= FALSE;
bStartlogin 	:= FALSE;
Serial_Use		:= FALSE;


SendSMS_Berror := FALSE ;
ReadSMS_bError := FALSE ;
LoginSMS_bError := FALSE ; 
DeletedSMS_Error := FALSE ; 
DeletedAllSMS_Error := FALSE ; 

RS_Reset(RESET1 := TRUE);
RS_Reset(RESET1 := FALSE);
Reset 			:= FALSE;
IN_Reset_OPC 		:= FALSE;
END_METHOD

METHOD M_Send
VAR_INPUT
END_VAR

CASE ETAPE_Send OF
	0://Etape d'entree
		IF NOT SendSMS_bBusy  AND NOT Serial_Use AND IN_DataSetFifo_SendSMS.nCount > 0 AND NOT LoginSMS_bBusy AND NOT LoginSMS_bError THEN  //Si serial libre et buffer contient plus d'une infos
			ReadAct:=FALSE;	
			Serial_Use:=TRUE;
			//bStartSend:=TRUE;
			SendSMS_bError := FALSE;
			Num_Tel := '';
			Message_Send:='';
			IN_DataSetFifo_SendSMS.A_Get();  //recuperation du message dans le send buffer 
			ETAPE_Send := 20  ; 
		ELSE
			ReadAct:=TRUE;	// En attente de lecture de mot d'alarme
		END_IF
			
		20:// Check les utilisateurs pour l'envoi des SMS 
			IF AX_Numtel[CPT] <> '' AND  AX_Subscribed[CPT] AND IN_DataSetFifo_SendSMS.out.Num_tel = '' AND (AX_User_LVL[CPT] AND IN_DataSetFifo_SendSMS.out.Alarms_LVL)>0    THEN
				// On envoi l'alarme si l'utilisateur est subscribed , et est dans la liste de diffusion de l'alarme
				Num_Tel:=AX_NumTel[CPT];
				bStartSend:=TRUE;
				ETAPE_Send:=1;
				MesTimeStamp := CONCAT(REPLACE(STR1:= IN_DataSetFifo_SendSMS.Out.TimeStamp_Act, STR2 := ' ', L := 1, P := 11), ' ') ;

				Message_Send := CONCAT(str1:=CONCAT(str1:=CONCAT(str1:=MesTimeStamp, str2:='$NID:' ), STR2:= UINT_TO_STRING(IN_DataSetFifo_SendSMS.out.ID)), STR2:=' ,' ) ; 
				Message_Send := CONCAT(STR1:=Message_Send , STR2:= IN_AX_Journal[IN_DataSetFifo_SendSMS.out.IndexWord][IN_DataSetFifo_SendSMS.Out.IndexBit].Message);
				
				IF IN_DataSetFifo_SendSMS.OUT.Active  THEN //Connaitre le statut de l'alarme: Active ou Non active
					Message_Send:=Concat(left(Message_Send, 125),' : Active');	// ajout de la mention activee ou desactive 
				ELSE
					Message_Send:=concat(left(Message_Send, 125),' : Desactive');
				END_IF
			ELSIF ( NOT AX_Subscribed[CPT] OR (AX_User_LVL[CPT] AND IN_DataSetFifo_SendSMS.out.Alarms_LVL)=0  ) AND IN_DataSetFifo_SendSMS.out.Num_tel = ''  THEN
				// L'alarme n'est pas envoyéeà cet utilisateur	
				Num_Tel := '';
				ETAPE_Send:=2;
			ELSIF IN_DataSetFifo_SendSMS.out.Num_tel <> ''  THEN
				// Si un numero de telephone est renseigné précisement, on envoi à ce numéro quelque soit la liste de diffusion , ou si l'utilisateur est subscribed
				bStartSend:=TRUE;
				Message_Send := CONCAT(STR1:=Message_Send , STR2:= IN_AX_Journal[IN_DataSetFifo_SendSMS.out.IndexWord][IN_DataSetFifo_SendSMS.Out.IndexBit].Message);
				Num_Tel:=IN_DataSetFifo_SendSMS.Out.Num_tel;
				ETAPE_Send:=1;
			ELSE
				// L'alarme n'est pas envoyée		
				Num_Tel := '';
				ETAPE_Send:=2;
			END_IF

	1://Envois du message
		Bstartsend:=FALSE;	
		IF NOT SendSMS_bBusy  THEN
			IF IN_DataSetFifo_SendSMS.OUT.IndexWord > 0 AND IN_DataSetFifo_SendSMS.In.Num_tel = ''   THEN
				ETAPE_Send:=2; // Alarme
				
			ELSE
				ETAPE_Send:=3; // Retour Sms ou utilisateur de renseignée
			END_IF
		ELSIF NOT SendSMS_bBusy AND SendSMS_Berror THEN // GGY
			//ETAPE_Send:=0; modif lWN seminaire 26/08/2020, gestion des ATE0, si erreur on supprime tout de meme le sms.
			ETAPE_Send:= 3;
			SendSMS_Berror := FALSE ; // On reset l'error apres avoir supprimé le SMS . 
			
		END_IF
		
	2:// Switch a un autre utilisateur
		IF CPT< CstNbUser THEN
			CPT:=CPT+1;
			ETAPE_Send:=20;
		ELSE
			ETAPE_Send:=3;
		END_IF
	
	3://Suppression de l'alarme et on passe au prochaine element dans le fifo
		IN_DataSetFifo_SendSMS.A_Remove();
		CPT:=1;
		Message_Send:='';
		ETAPE_Send:=0;
		Serial_Use:=FALSE;
		bStartSend:=FALSE;

END_CASE
END_METHOD

END_PROGRAM

// ---- 00_FunctionsBlocks/Beckhoff/Fifo/FB_SMSDatasetFifo_Read.TcPOU
FUNCTION_BLOCK FB_SMSDatasetFifo_Read
VAR_INPUT
    bOverwrite : BOOL;
    In         : ST_SMSDataSetEntry_Read;
END_VAR
VAR_OUTPUT
    bOk        : BOOL;
    nCount     : UDINT;
    nLoad      : UDINT;
    Out        : ST_SMSDataSetEntry_Read;
END_VAR
VAR
    arrBuffer  : ARRAY[0..Max_buffer_size_G] OF BYTE; (* Buffer memory used by FB_MemRingBuffer function block *)
    fbBuffer   : FB_MemRingBuffer;
END_VAR

ACTION A_Add:
fbBuffer.A_AddTail(pWrite := ADR(in),
						   cbWrite:=SIZEOF(in),
						   pBuffer:=ADR(arrBuffer),
						   cbBuffer:=SIZEOF(arrBuffer),
						   bOK=>bOK,
						   nCount =>nCount);
IF NOT bOK THEN 
	IF bOverwrite THEN
		fbBuffer.A_RemoveHead();(*remove one oldest entry*)
		fbBuffer.A_AddTail(bOK => bOk,nCount => nCount);
	END_IF
END_IF

nload := (fbbuffer.cbSize * 100)/(Max_buffer_size_G);
END_ACTION

ACTION A_Get:
fbBuffer.A_GetHead(pWrite := ADR(out),
						   cbWrite:=SIZEOF(out),
						   pBuffer:=ADR(arrBuffer),
						   cbBuffer:=SIZEOF(arrBuffer),
						   bOK=>bOK,
						   nCount =>nCount);
nload := (fbbuffer.cbSize * 100)/(Max_buffer_size_G);
END_ACTION

ACTION A_Remove:
fbBuffer.A_RemoveHead(pRead:=ADR(out),
						cbRead:=SIZEOF(out),
						pBuffer:=ADR(arrBuffer),
						cbBuffer:=SIZEOF(arrBuffer),
						bOK=>bOK,
						nCount =>nCount);
nload := (fbbuffer.cbSize * 100)/(Max_buffer_size_G);
END_ACTION

ACTION A_Reset:
MEMSET(ADR(arrBuffer),0,SIZEOF(arrBuffer)); (*reset internal buffer*)
fbBuffer.A_Reset(bOK=>bOK,nCount=>ncount);
nload := (fbbuffer.cbSize * 100)/(Max_buffer_size_G);
END_ACTION

END_FUNCTION_BLOCK

// ---- 00_FunctionsBlocks/Beckhoff/Fifo/FB_SMSDatasetFifo_Send.TcPOU
FUNCTION_BLOCK FB_SMSDatasetFifo_Send
VAR_INPUT
    bOverwrite : BOOL;
    In         : ST_SMSDataSetEntry_Send;
END_VAR
VAR_OUTPUT
    bOk        : BOOL;
    nCount     : UDINT;
    nLoad      : UDINT;
    Out        : ST_SMSDataSetEntry_Send;
END_VAR
VAR
    arrBuffer  : ARRAY[0..Max_buffer_size_G] OF BYTE; (* Buffer memory used by FB_MemRingBuffer function block *)
    fbBuffer   : FB_MemRingBuffer;
END_VAR

ACTION A_Add:
fbBuffer.A_AddTail(pWrite := ADR(in),
						   cbWrite:=SIZEOF(in),
						   pBuffer:=ADR(arrBuffer),
						   cbBuffer:=SIZEOF(arrBuffer),
						   bOK=>bOK,
						   nCount =>nCount);
IF NOT bOK THEN 
	IF bOverwrite THEN
		fbBuffer.A_RemoveHead();(*remove one oldest entry*)
		fbBuffer.A_AddTail(bOK => bOk,nCount => nCount);
	END_IF
END_IF

nload := (fbbuffer.cbSize * 100)/(Max_buffer_size_G);
END_ACTION

ACTION A_Get:
fbBuffer.A_GetHead(pWrite := ADR(out),
						   cbWrite:=SIZEOF(out),
						   pBuffer:=ADR(arrBuffer),
						   cbBuffer:=SIZEOF(arrBuffer),
						   bOK=>bOK,
						   nCount =>nCount);
nload := (fbbuffer.cbSize * 100)/(Max_buffer_size_G);
END_ACTION

ACTION A_Remove:
fbBuffer.A_RemoveHead(pRead:=ADR(out),
						cbRead:=SIZEOF(out),
						pBuffer:=ADR(arrBuffer),
						cbBuffer:=SIZEOF(arrBuffer),
						bOK=>bOK,
						nCount =>nCount);
nload := (fbbuffer.cbSize * 100)/(Max_buffer_size_G);
END_ACTION

ACTION A_Reset:
MEMSET(ADR(arrBuffer),0,SIZEOF(arrBuffer)); (*reset internal buffer*)
fbBuffer.A_Reset(bOK=>bOK,nCount=>ncount);
nload := (fbbuffer.cbSize * 100)/(Max_buffer_size_G);
END_ACTION

END_FUNCTION_BLOCK

// ---- 00_FunctionsBlocks/Beckhoff/Communication/SMS/FB_ReadSMS.TcPOU
FUNCTION_BLOCK FB_ReadSMS

VAR_INPUT PERSISTENT 
	ParamTimeoutReadSMS		: TIME := T#3S ; // Tiemout pour lire les sms.  Attention , ce parametre est très important . Si pas assez grand, risque de données tronquées. 
	
	
	
END_VAR

VAR_INPUT
	bStart					: BOOL;
	nIndex					: USINT;
	
END_VAR
VAR_OUTPUT
	sMessageText			: STRING(240);
	bBusy					: BOOL;
	bError					: BOOL;
	nErrorID				: UINT;
	
END_VAR

VAR_IN_OUT
	stTxBuffer				: ComBuffer;
	stRxBuffer				: ComBuffer;
END_VAR

VAR
	rtrigStart				: R_TRIG;

	fbSendData				: SendData;
	fbReceiveData			: ReceiveData;
	fbClearComBuffer		: ClearComBuffer;

	i,iSavedIndex			: INT;
	uiAnalyzeAnswer			: UINT;
	nStep					: UINT; (* sequence state *)
	tonWaitTime				: TON;
	tonTimeOut				: TON;
	tTimeout				: TIME:=T#30S;


	arAnswerOK				: ARRAY[1..2] OF BYTE:=[16#4F,16#4B];
	arAnswerErr				: ARRAY[1..5] OF BYTE:=[16#45,16#52,16#52,16#4F,16#52];

	sReadSMS				: STRING(15);			(*Command-String*)
	arReadSMS				: ARRAY[1..15] OF BYTE; (*Command-ARRAY*)
	arReadSMSAnswerRcv		: ARRAY[1..300] OF BYTE;(*Received answer of the command*)
	arReadSMSAnswerClr		: ARRAY[1..300] OF BYTE;(*Empty-ARRAY to clear the answer for debugging*)
END_VAR


	rtrigStart(CLK:=bStart);

	tonTimeout();
	IF (tonTimeout.Q) THEN
		tonTimeout(IN := FALSE);
		nStep := 900;
	END_IF


	CASE nStep OF

	0: 	(*Idle Step*);
		MEMSET(ADR(sMessageText),0,SIZEOF(sMessageText));
		tonTimeout(IN:=FALSE);
		IF (rtrigStart.Q AND NOT bBusy) THEN
			nStep := 5;
			bBusy := TRUE;
			
		ELSE
			bBusy := FALSE;
		END_IF


	5:
		bError					:= FALSE;
		nErrorId				:= 0;
		tonWaitTime				(IN := FALSE);
		tonTimeout				(IN := TRUE, PT := tTimeout);
		fbClearComBuffer		(buffer:=stRxBuffer);
		fbClearComBuffer		(buffer:=stTxBuffer);
		sMessageText			:= '';
		MEMSET(ADR(sMessageText),0,SIZEOF(sMessageText));
		nStep := 50;


	50:(*Create command-Arrays*)
		(*Read SMS*)
		sReadSMS:='AT+CMGR="';
		sReadSMS:=CONCAT(sReadSMS,USINT_TO_STRING(nIndex));
		sReadSMS:=CONCAT(sReadSMS,'"X');	(*The "X" is a placeholder in the send-string
											for the "CR" (Hex 0D) in the send-Array*)
		MEMCPY(ADR(arReadSMS),ADR(sReadSMS),LEN(sReadSMS)); (*Copy String to ARRAY*)
		arReadSMS[LEN(sReadSMS)]:=16#0D;	(*Place the "CR" in the array*)

		nStep	:= 100;


	100:(*Send read-command*)
		fbSendData(
		pSendData:=ADR(arReadSMS),
		Length:= LEN(sReadSMS),
		TXbuffer:= stTxBuffer);

		IF NOT fbSendData.Busy THEN
			nStep:=110;
		END_IF

		IF  fbSendData.Error<>0 THEN
			bError:= TRUE;
			nErrorID:= fbSendData.Error;
			nStep:=1000;
		END_IF


	110:(*The beginning and the contents of the answer can vary. If the message-slot contains
		a valid message	it begins with "+CMGR" and ends with "OK". 
		An answer of an empty slot is only "OK". In case of an error the answer is only "ERROR"
		So there is no proper prefix to wait fOR *)
		fbReceiveData(
		pPrefix:= 0,
		LenPrefix:= 0,
		pReceiveData:= ADR(arReadSMSAnswerRcv),
		SizeReceiveData:= SIZEOF(arReadSMSAnswerRcv),
		Timeout:= ParamTimeoutReadSMS ,		
		RXbuffer:= stRxBuffer);

		(*Telegram is received*)
		IF 			fbReceiveData.DataReceived
			AND NOT fbReceiveData.busy	THEN
						nStep:=120;
		END_IF


	120:(* NEW VERSION  : ON recupère la commande si elle est non vide ou non pleine. on analyze les champs ensuite.*)

		(* OLD VERSION  : Find an "OK" or an "ERROR"-Part in the answer
		Search from the end of the received string to the top and take the first match
		not to get a SMS-written "ok" or "error"*)
		uiAnalyzeAnswer	:=0;
		iSavedIndex		:=0;
		IF arReadSMSAnswerRcv[SIZEOF(arReadSMSAnswerRcv)]<> 0 THEN		
			nErrorID := 16#FFFF; // La taille du message dépasse ce que l'on peut récupérer
		ELSIF arReadSMSAnswerRcv[1]= 0 THEN 
			nErrorID := 16#800E; // Le message est vide 
		ELSE
			
			FOR i:= UINT_TO_INT(SIZEOF(arReadSMSAnswerRcv)) TO 1 BY -1 DO		// i:= uint_to_int(SIZEOF(arReadSMSAnswerRcv)-5) TO 1 BY -1 DO	
				IF 		arReadSMSAnswerRcv[i]	<> 0 THEN 	//= arAnswerOK[1] AND arReadSMSAnswerRcv[i+1] 	= arAnswerOK[2]		THEN
						
						iSavedIndex:=i;// iSavedIndex:=i-1;
						
						IF iSavedIndex > 2 THEN 
							uiAnalyzeAnswer:=1;		(*Read SMS successfully executed*)
						ELSE
							uiAnalyzeAnswer:=0;		(*Read SMS successfully executed*)
							nErrorID := 16#FFFF; // La taille du message est inférieru à deux word , on ne peut pas le copier dans un string
						END_IF
						
					EXIT;
	(*
				ELSIF	arReadSMSAnswerRcv[i]		= arAnswerErr[1]
					AND arReadSMSAnswerRcv[i+1] 	= arAnswerErr[2]
					AND arReadSMSAnswerRcv[i+2] 	= arAnswerErr[3]
					AND arReadSMSAnswerRcv[i+3] 	= arAnswerErr[4]
					AND arReadSMSAnswerRcv[i+4] 	= arAnswerErr[5]	THEN
						uiAnalyzeAnswer:=2;		(*Read SMS failed*)
					EXIT;
					*)
				END_IF
			END_FOR
			
		END_IF
		CASE uiAnalyzeAnswer OF
			0:(*Undefined Answer*)
				bError:= TRUE;
				//nErrorID:= 16#800E;
				nStep:=1000;
				//nStep:=1000;

			1:(*Read SMS successfully executed*)
				nStep:=130;

			2:(*Read SMS failed*)
				bError:= TRUE;
				nErrorID:= 16#800D;
				nStep:=1000;
		END_CASE


	130:(*Copy message-Array to String*)
		MEMCPY(ADR(sMessageText),(ADR(arReadSMSAnswerRcv)+2),(iSavedIndex)); (*"2" : Do not read the first two digits of the answer. It always begins with "0D,0A"*)

		IF (FIND(sMessageText,'ERROR')>0) THEN 
			// Il y a une erreru dans la lecture du message. 
			bError := TRUE ; 
			nErrorID:= 16#800D;
			nStep:=1000;
		ELSE 
			nStep:=1000;
		END_IF



	900:(*Timeout*)
		bError:= TRUE;
		nErrorID:= 16#8001;
		nStep:=1000;


	1000:(*Reset Receive-FB*)
		fbReceiveData(	Reset:=TRUE,RXbuffer:= stRxBuffer);
		tonWaitTime(IN:=TRUE, PT:=t#500ms);
		IF	tonWaitTime.Q	THEN
			fbReceiveData(	Reset:=FALSE,RXbuffer:= stRxBuffer);
			nStep:=1010;
		END_IF


	1010:(*Send/Receive successful -> Reset FBs*)
		fbClearComBuffer(buffer:=stRxBuffer);
		fbClearComBuffer(buffer:=stTxBuffer);
		arReadSMSAnswerRcv	:= arReadSMSAnswerClr;
		nStep:=0;
		bBusy:=FALSE;

	END_CASE;

END_FUNCTION_BLOCK

// ---- 00_FunctionsBlocks/Beckhoff/Communication/SMS/FB_SendSMS.TcPOU
FUNCTION_BLOCK FB_SendSMS

VAR_INPUT
	bStart					: BOOL;  			(* Rising edge start fb execution *)
	sPhoneNumber			: STRING(30);		(* phone Number *)
	sSMSText				: T_MaxString;		(* Message Text *)
	bReset					: BOOL ; 
END_VAR

VAR_OUTPUT
	bBusy					: BOOL;
	bError					: BOOL;
	nErrorID				: UINT;
	
END_VAR

VAR_IN_OUT
	stTxBuffer				: ComBuffer;
	stRxBuffer				: ComBuffer;
	
END_VAR

VAR
	rtrigStart				: R_TRIG;

	fbSendData				: SendData;
	fbReceiveData			: ReceiveData;
	fbClearComBuffer		: ClearComBuffer;

	i						: UINT;
	uiAnalyzeAnswer			: UINT;
	nStep					: UINT; (* sequence state *)
	tonWaitTime				: TON;
	tonTimeOut				: TON;
	tTimeout				: TIME:=T#60S;

	byAnswerEnter			: BYTE:=16#3E; //">"
	arAnswerCMGS			: ARRAY[1..4] OF BYTE:=[16#43,16#4D,16#47,16#53]; //CMGS
	arAnswerOK				: ARRAY[1..2] OF BYTE:=[16#4F,16#4B]; //OK
	arAnswerErr				: ARRAY[1..5] OF BYTE:=[16#45,16#52,16#52,16#4F,16#52]; //ERROR

	sSetSMSFormat			: STRING(10);			(*Command-String*)
	arSetSMSFormat			: ARRAY[1..10] OF BYTE;	(*Command-ARRAY*)
	arSetSMSFormatAnswerRcv	: ARRAY[1..5] OF BYTE;	(*Received answer of the command*)
	arSetSMSFormatAnswerClr	: ARRAY[1..5] OF BYTE;	(*Empty-ARRAY to clear the answer for debugging*)

	sSendSMSPart1			: STRING(40);			(*Command-String*)
	arSendSMSPart1			: ARRAY[1..40] OF BYTE;	(*Command-ARRAY*)
	arSendSMSPart1AnswerRcv	: ARRAY[1..5] OF BYTE;	(*Received answer of the command*)
	arSendSMSPart1AnswerClr	: ARRAY[1..5] OF BYTE;	(*Empty-ARRAY to clear the answer for debugging*)

	sSendSMSPart2			: STRING(170);			(*Command-String*)
	arSendSMSPart2			: ARRAY[1..170] OF BYTE;(*Command-ARRAY*)
	arSendSMSPart2AnswerRcv	: ARRAY[1..35] OF BYTE;	(*Received answer of the command*)
	arSendSMSPart2AnswerClr	: ARRAY[1..35] OF BYTE;	(*Empty-ARRAY to clear the answer for debugging*)
END_VAR


IF bReset THEN 
	bError := FALSE ; 
	bReset:= FALSE ; 
END_IF


	rtrigStart(CLK:=bStart);

	tonTimeout();
	IF (tonTimeout.Q) THEN
		tonTimeout(IN := FALSE);
		nStep := 900;
	END_IF


	CASE nStep OF

	0:	(*Idle Step*);
		tonTimeout(IN:=FALSE);
		IF (rtrigStart.Q AND NOT bBusy) THEN
			nStep := 5;
			bBusy := TRUE;
		ELSE
			bBusy := FALSE;
		END_IF


	5:
		bError					:= FALSE;
		nErrorId				:= 0;
		tonWaitTime				(IN := FALSE);
		tonTimeout				(IN := TRUE, PT := tTimeout);
		fbClearComBuffer		(buffer:=stRxBuffer);
		fbClearComBuffer		(buffer:=stTxBuffer);
		arSetSMSFormatAnswerRcv	:= arSetSMSFormatAnswerClr;
		arSendSMSPart1AnswerRcv	:= arSendSMSPart1AnswerClr;
		arSendSMSPart2AnswerRcv	:= arSendSMSPart2AnswerClr;
	
		nStep := 10;


	10:(*Length of phone-number within limits?*)
		IF 		LEN(sPhoneNumber) < 1
			OR	LEN(sPhoneNumber) > 25 THEN
			bError		:= TRUE;
			nErrorID	:= 16#8006;
			nStep		:= 1000;
		ELSE
			nStep		:= 20;
		END_IF


	20:(*Phone-number contains correct characters? 0..9, + *)
		FOR i:=1 TO LEN(sPhoneNumber) DO
			IF 	((ASC(MID(sPhoneNumber,1,i)) < 16#30) OR (ASC(MID(sPhoneNumber,1,i)) > 16#39))
				AND NOT (ASC(MID(sPhoneNumber,1,i)) = 16#2B)	THEN
				bError		:= TRUE;	(*a non-numeric character in the phone-number, except the "+"-sign*)
				nErrorID	:= 16#8007;
			END_IF
		END_FOR

		IF bError	THEN
			nStep	:= 1000;
		ELSE
			nStep	:= 30;
		END_IF


	30:(*Length of SMS-Text within limits?*)
		IF 	(LEN(sSMSText) < 1 OR LEN(sSMSText) > 160) THEN
			bError		:= TRUE;
			nErrorID	:= 16#8008;
			nStep		:= 1000;
		ELSE
			nStep		:= 50;
		END_IF


	50:(*Create command-Arrays*)

		(*Set SMS Format to textmode*)
		sSetSMSFormat:='AT+CMGF=1';
		sSetSMSFormat:=CONCAT(sSetSMSFormat,'X');	(*The "X" is a placeholder in the send-string
													for the "CR" (Hex 0D) in the send-Array*)
		MEMCPY(ADR(arSetSMSFormat),ADR(sSetSMSFormat),LEN(sSetSMSFormat)); (*Copy String to ARRAY*)
		arSetSMSFormat[LEN(sSetSMSFormat)]:=16#0D;	(*Place the "CR" in the array*)


		(*Send SMS, Part1 - Phone-number*)
		sSendSMSPart1:='AT+CMGS="';
		sSendSMSPart1:=CONCAT(sSendSMSPart1,sPhoneNumber);
		sSendSMSPart1:=CONCAT(sSendSMSPart1,'"X');	(*The "X" is a placeholder in the send-string
													for the "CR" (Hex 0D) in the send-Array*)
		MEMCPY(ADR(arSendSMSPart1),ADR(sSendSMSPart1),LEN(sSendSMSPart1)); (*Copy String to ARRAY*)
		arSendSMSPart1[LEN(sSendSMSPart1)]:=16#0D;	(*Place the "CR" in the array*)


		(*Send SMS, Part2 - text*)
		sSendSMSPart2:='"';
		sSendSMSPart2:=CONCAT(sSendSMSPart2,sSMSText);
		sSendSMSPart2:=CONCAT(sSendSMSPart2,'"X');	(*The "X" is a placeholder in the send-string
													for the "ctrl+z" (Hex 1A) in the send-Array*)
		MEMCPY(ADR(arSendSMSPart2),ADR(sSendSMSPart2),LEN(sSendSMSPart2)); (*Copy String to ARRAY*)
		arSendSMSPart2[LEN(sSendSMSPart2)]:=16#1A;	(*Place the "ctrl+z" in the array*)


		nStep	:= 100;


	100:(*Set SMS-Format to text-Mode*)
		fbSendData(
		pSendData:=ADR(arSetSMSFormat),
		Length:= LEN(sSetSMSFormat),
		TXbuffer:= stTxBuffer);

		IF NOT fbSendData.Busy THEN
			nStep:=110;
		END_IF

		IF  fbSendData.Error<>0 THEN
			bError:= TRUE;
			nErrorID:= fbSendData.Error;
			nStep:=1000;
		END_IF


	110:(*Wait for OK or Err-Answer. Any other answer caused by Comm-Error will end in global timeout*)
		fbReceiveData(
		pPrefix:= 0,
		LenPrefix:= 0,
		pReceiveData:= ADR(arSetSMSFormatAnswerRcv),
		SizeReceiveData:= SIZEOF(arSetSMSFormatAnswerRcv),
		Timeout:= t#500ms,
		RXbuffer:= stRxBuffer);

		(*Telegram is received*)
		IF 			fbReceiveData.DataReceived
			AND NOT fbReceiveData.busy	THEN
						nStep:=120;
		END_IF


	120:(*Analyze answer*)
		IF		(arSetSMSFormatAnswerRcv[3]=arAnswerOK[1]) AND (arSetSMSFormatAnswerRcv[4]=arAnswerOK[2])	THEN
					nStep:=200;			(*Set-format successfully executed*)
		ELSIF	(arSetSMSFormatAnswerRcv[3]=arAnswerErr[1]) AND (arSetSMSFormatAnswerRcv[4]=arAnswerErr[2])	THEN
					bError:= TRUE;
					nErrorID:= 16#8009;	(*Set-format failed*)
					nStep:=1000;
		ELSE
					bError:= TRUE;
					nErrorID:= 16#800A;	(*Undefined answer*)
					nStep:=1000;
		END_IF


	200:(*Send SMS Part1 - Command and phone-number*)
		fbSendData(
		pSendData:=ADR(arSendSMSPart1),
		Length:= LEN(sSendSMSPart1),
		TXbuffer:= stTxBuffer);

		IF NOT fbSendData.Busy THEN
			nStep:=210;
		END_IF

		IF  fbSendData.Error<>0 THEN
			bError:= TRUE;
			nErrorID:= fbSendData.Error;
			nStep:=1000;
		END_IF


	210:(*Wait explicitly for an ">"-Answer because normally only ">" is possible,
		any other answer is regarded faulty and will end in global timeout*)

		fbReceiveData(
		pPrefix:= ADR(byAnswerEnter),
		LenPrefix:= 1,
		pReceiveData:= ADR(arSendSMSPart1AnswerRcv),
		SizeReceiveData:= SIZEOF(arSendSMSPart1AnswerRcv),
		Timeout:= t#500ms,
		Reset:= FALSE,
		RXbuffer:= stRxBuffer);

		(*Telegram is received*)
		IF 			fbReceiveData.DataReceived
			AND NOT fbReceiveData.busy			THEN
						nStep:=220;
		END_IF


	220:(*Send SMS Part2 - text-part*)
		fbSendData(
		pSendData:=ADR(arSendSMSPart2),
		Length:= LEN(sSendSMSPart2),
		TXbuffer:= stTxBuffer);

		IF NOT fbSendData.Busy THEN
			nStep:=230;
		END_IF

		IF  fbSendData.Error<>0 THEN
			bError:= TRUE;
			nErrorID:= fbSendData.Error;
			nStep:=1000;
		END_IF


	230:(*Wait explicitly for a "CMGS"-Answer because normally only "CMGS" is possible,
		any other answer is regarded faulty and will end in global timeout*)
		fbReceiveData(
		pPrefix:= ADR(arAnswerCMGS),
		LenPrefix:= SIZEOF(arAnswerCMGS),
		pReceiveData:= ADR(arSendSMSPart2AnswerRcv),
		SizeReceiveData:= SIZEOF(arSendSMSPart2AnswerRcv),
		Timeout:= t#1000ms,
		RXbuffer:= stRxBuffer);

		(*Telegram is received*)
		IF 			fbReceiveData.DataReceived
			AND NOT fbReceiveData.busy	THEN
						nStep:=240;
		END_IF


	240:(*Find an "OK" or an "ERROR"-Part in the answer*)
		uiAnalyzeAnswer:=0;
		FOR i:= 1 TO (SIZEOF(arSendSMSPart2AnswerRcv)-5) DO
			IF 		arSendSMSPart2AnswerRcv[i]		= arAnswerOK[1]
				AND arSendSMSPart2AnswerRcv[i+1] 	= arAnswerOK[2]		THEN
					uiAnalyzeAnswer:=1;		(*Send SMS successfully executed*)
					EXIT;

			ELSIF	arSendSMSPart2AnswerRcv[i]		= arAnswerErr[1]
				AND arSendSMSPart2AnswerRcv[i+1] 	= arAnswerErr[2]
				AND arSendSMSPart2AnswerRcv[i+2] 	= arAnswerErr[3]
				AND arSendSMSPart2AnswerRcv[i+3] 	= arAnswerErr[4]
				AND arSendSMSPart2AnswerRcv[i+4] 	= arAnswerErr[5]	THEN
					uiAnalyzeAnswer:=2;		(*Send SMS failed*)
					EXIT;
			END_IF
		END_FOR

		CASE uiAnalyzeAnswer OF
			0:(*Undefined Answer*)
				bError:= TRUE;
				nErrorID:= 16#800D;
				nStep:=1000;

			1:(*Send SMS successfully executed*)
				nStep:=1000;

			2:(*Send SMS failed*)
				bError:= TRUE;
				nErrorID:= 16#800C;
				nStep:=1000;
		END_CASE


	900:(*Timeout*) // delete last sms in case of timeout
		bError:= TRUE;
		nErrorID:= 16#8001;
		nStep:=1000;


	1000:(*Reset Receive-FB*)
		fbReceiveData(	Reset:=TRUE,RXbuffer:= stRxBuffer);
		tonWaitTime(IN:=TRUE, PT:=t#500ms);
		IF	tonWaitTime.Q	THEN
			fbReceiveData(	Reset:=FALSE,RXbuffer:= stRxBuffer);
			nStep:=1010;
		END_IF


	1010:	(*Send/Receive successful -> Reset FBs*)
		fbClearComBuffer(buffer:=stRxBuffer);
		fbClearComBuffer(buffer:=stTxBuffer);
		nStep:=0;
		bBusy:=FALSE;

	END_CASE;

END_FUNCTION_BLOCK

// ---- 00_FunctionsBlocks/Beckhoff/Communication/SMS/FB_DeleteSMS.TcPOU
FUNCTION_BLOCK FB_DeleteSMS
VAR_INPUT
	bStart					: BOOL;
	nIndex					: USINT;
END_VAR
VAR_OUTPUT
	bBusy					: BOOL;
	bError					: BOOL;
	nErrorID				: UINT;
END_VAR

VAR_IN_OUT
	stTxBuffer				: ComBuffer;
	stRxBuffer				: ComBuffer;
END_VAR

VAR
	rtrigStart				: R_TRIG;

	fbSendData				: SendData;
	fbReceiveData			: ReceiveData;
	fbClearComBuffer		: ClearComBuffer;

	i						: INT;
	uiAnalyzeAnswer			: UINT;
	nStep					: UINT; (* sequence state *)
	tonWaitTime				: TON;
	tonTimeOut				: TON;
	tTimeout				: TIME:=t#5s;

	arAnswerOK				: ARRAY[1..2] OF BYTE:=[16#4F,16#4B];
	arAnswerErr				: ARRAY[1..5] OF BYTE:=[16#45,16#52,16#52,16#4F,16#52];

	sDeleteSMS				: STRING(15);			(*Command-String*)
	arDeleteSMS				: ARRAY[1..15] OF BYTE; (*Command-ARRAY*)
	arDeleteSMSAnswerRcv	: ARRAY[1..200] OF BYTE;(*Received answer of the command*)
	arDeleteSMSAnswerClr	: ARRAY[1..200] OF BYTE;(*Empty-ARRAY to clear the answer for debugging*)
END_VAR


	rtrigStart(CLK:=bStart);

	tonTimeout();
	IF (tonTimeout.Q) THEN
		tonTimeout(IN := FALSE);
		nStep := 900;
	END_IF


	CASE nStep OF

	0: 	(*Idle Step*);
		tonTimeout(IN:=FALSE);
		IF (rtrigStart.Q AND NOT bBusy) THEN
			nStep := 5;
			bBusy := TRUE;
		ELSE
			bBusy := FALSE;
		END_IF


	5:
		bError					:= FALSE;
		nErrorId				:= 0;
		tonWaitTime				(IN := FALSE);
		tonTimeout				(IN := TRUE, PT := tTimeout);
		fbClearComBuffer		(buffer:=stRxBuffer);
		fbClearComBuffer		(buffer:=stTxBuffer);
		arDeleteSMSAnswerRcv	:= arDeleteSMSAnswerClr;

		nStep := 50;


	50:(*Create command-Arrays*)

		(*Delete-command*)
		sDeleteSMS:='AT+CMGD="';
		sDeleteSMS:=CONCAT(sDeleteSMS,USINT_TO_STRING(nIndex));
		sDeleteSMS:=CONCAT(sDeleteSMS,'"X');	(*The "X" is a placeholder in the send-string
												for the "CR" (Hex 0D) in the send-Array*)
		MEMCPY(ADR(arDeleteSMS),ADR(sDeleteSMS),LEN(sDeleteSMS)); (*Copy String to ARRAY*)
		arDeleteSMS[LEN(sDeleteSMS)]:=16#0D;	(*Place the "CR" in the array*)

		nStep	:= 100;


	100:(*Send delete-command*)
		fbSendData(
		pSendData:=ADR(arDeleteSMS),
		Length:= LEN(sDeleteSMS),
		TXbuffer:= stTxBuffer);

		IF NOT fbSendData.Busy THEN
			nStep:=110;
		END_IF

		IF  fbSendData.Error<>0 THEN
			bError:= TRUE;
			nErrorID:= fbSendData.Error;
			nStep:=1000;
		END_IF


	110:(*Wait for the answer*)
		fbReceiveData(
		pPrefix:= 0,
		LenPrefix:= 0,
		pReceiveData:= ADR(arDeleteSMSAnswerRcv),
		SizeReceiveData:= SIZEOF(arDeleteSMSAnswerRcv),
		Timeout:= t#1000ms,
		RXbuffer:= stRxBuffer);

		(*Telegram is received*)
		IF 			fbReceiveData.DataReceived
			AND NOT fbReceiveData.busy	THEN
						nStep:=120;
		END_IF


	120:(*Find an "OK" or an "ERROR"-Part in the answer*)
		uiAnalyzeAnswer	:=0;
		FOR i:= (SIZEOF(arDeleteSMSAnswerRcv)-5) TO 1 BY -1 DO
			IF 		arDeleteSMSAnswerRcv[i]		= arAnswerOK[1]
				AND arDeleteSMSAnswerRcv[i+1] 	= arAnswerOK[2]		THEN
					uiAnalyzeAnswer:=1;		(*Delete SMS successfully executed*)
				EXIT;

			ELSIF	arDeleteSMSAnswerRcv[i]		= arAnswerErr[1]
				AND arDeleteSMSAnswerRcv[i+1] 	= arAnswerErr[2]
				AND arDeleteSMSAnswerRcv[i+2] 	= arAnswerErr[3]
				AND arDeleteSMSAnswerRcv[i+3] 	= arAnswerErr[4]
				AND arDeleteSMSAnswerRcv[i+4] 	= arAnswerErr[5]	THEN
					uiAnalyzeAnswer:=2;		(*Delete SMS failed*)
				EXIT;
			END_IF
		END_FOR

		CASE uiAnalyzeAnswer OF
			0:(*Undefined Answer*)
				bError:= TRUE;
				nErrorID:= 16#8010;
				nStep:=1000;

			1:(*Delete SMS successfully executed*)
				nStep:=1000;

			2:(*Delete SMS failed*)
				bError:= TRUE;
				nErrorID:= 16#800F;
				nStep:=1000;
		END_CASE


	900:(*Timeout*)
		bError:= TRUE;
		nErrorID:= 16#8001;
		nStep:=1000;


	1000:(*Reset Receive-FB*)
		fbReceiveData(	Reset:=TRUE,RXbuffer:= stRxBuffer);
		tonWaitTime(IN:=TRUE, PT:=t#500ms);
		IF	tonWaitTime.Q	THEN
			fbReceiveData(	Reset:=FALSE,RXbuffer:= stRxBuffer);
			nStep:=1010;
		END_IF


	1010:(*Send/Receive successful -> Reset FBs*)
		fbClearComBuffer(buffer:=stRxBuffer);
		fbClearComBuffer(buffer:=stTxBuffer);
		nStep:=0;
		bBusy:=FALSE;

	END_CASE;

END_FUNCTION_BLOCK

// ---- 00_FunctionsBlocks/Beckhoff/Communication/SMS/FB_DeleteAllSMS.TcPOU
FUNCTION_BLOCK FB_DeleteAllSMS
VAR_INPUT
	bStart					: BOOL;
END_VAR
VAR_OUTPUT
	bBusy					: BOOL;
	bError					: BOOL;
	nErrorID				: UINT;
END_VAR

VAR_IN_OUT
	stTxBuffer				: ComBuffer;
	stRxBuffer				: ComBuffer;
END_VAR

VAR
	rtrigStart				: R_TRIG;

	fbSendData				: SendData;
	fbReceiveData			: ReceiveData;
	fbClearComBuffer		: ClearComBuffer;

	i						: INT;
	uiAnalyzeAnswer			: UINT;
	nStep					: UINT; (* sequence state *)
	tonWaitTime				: TON;
	tonTimeOut				: TON;
	tTimeout				: TIME:=t#5s;

	arAnswerOK				: ARRAY[1..2] OF BYTE:=[16#4F,16#4B];
	arAnswerErr				: ARRAY[1..5] OF BYTE:=[16#45,16#52,16#52,16#4F,16#52];

	sDeleteSMS				: STRING(15);			(*Command-String*)
	arDeleteSMS				: ARRAY[1..15] OF BYTE; (*Command-ARRAY*)
	arDeleteSMSAnswerRcv	: ARRAY[1..200] OF BYTE;(*Received answer of the command*)
	arDeleteSMSAnswerClr	: ARRAY[1..200] OF BYTE;(*Empty-ARRAY to clear the answer for debugging*)
END_VAR


	rtrigStart(CLK:=bStart);

	tonTimeout();
	IF (tonTimeout.Q) THEN
		tonTimeout(IN := FALSE);
		nStep := 900;
	END_IF


	CASE nStep OF

	0: 	(*Idle Step*);
		tonTimeout(IN:=FALSE);
		IF (rtrigStart.Q AND NOT bBusy) THEN
			nStep := 5;
			bBusy := TRUE;
		ELSE
			bBusy := FALSE;
		END_IF


	5:
		bError					:= FALSE;
		nErrorId				:= 0;
		tonWaitTime				(IN := FALSE);
		tonTimeout				(IN := TRUE, PT := tTimeout);
		fbClearComBuffer		(buffer:=stRxBuffer);
		fbClearComBuffer		(buffer:=stTxBuffer);
		arDeleteSMSAnswerRcv	:= arDeleteSMSAnswerClr;

		nStep := 50;


	50:(*Create command-Arrays*)

		(*Delete-command*)
		sDeleteSMS:='AT+CMGD="';
		sDeleteSMS:=CONCAT(sDeleteSMS,'1,4');
		
		sDeleteSMS:=CONCAT(sDeleteSMS,'"X');	(*The "X" is a placeholder in the send-string
												for the "CR" (Hex 0D) in the send-Array*)
		MEMCPY(ADR(arDeleteSMS),ADR(sDeleteSMS),LEN(sDeleteSMS)); (*Copy String to ARRAY*)
		arDeleteSMS[LEN(sDeleteSMS)]:=16#0D;	(*Place the "CR" in the array*)

		nStep	:= 100;


	100:(*Send delete-command*)
		fbSendData(
		pSendData:=ADR(arDeleteSMS),
		Length:= LEN(sDeleteSMS),
		TXbuffer:= stTxBuffer);

		IF NOT fbSendData.Busy THEN
			nStep:=110;
		END_IF

		IF  fbSendData.Error<>0 THEN
			bError:= TRUE;
			nErrorID:= fbSendData.Error;
			nStep:=1000;
		END_IF


	110:(*Wait for the answer*)
		fbReceiveData(
		pPrefix:= 0,
		LenPrefix:= 0,
		pReceiveData:= ADR(arDeleteSMSAnswerRcv),
		SizeReceiveData:= SIZEOF(arDeleteSMSAnswerRcv),
		Timeout:= t#1000ms,
		RXbuffer:= stRxBuffer);

		(*Telegram is received*)
		IF 			fbReceiveData.DataReceived
			AND NOT fbReceiveData.busy	THEN
						nStep:=120;
		END_IF


	120:(*Find an "OK" or an "ERROR"-Part in the answer*)
		uiAnalyzeAnswer	:=0;
		FOR i:= (SIZEOF(arDeleteSMSAnswerRcv)-5) TO 1 BY -1 DO
			IF 		arDeleteSMSAnswerRcv[i]		= arAnswerOK[1]
				AND arDeleteSMSAnswerRcv[i+1] 	= arAnswerOK[2]		THEN
					uiAnalyzeAnswer:=1;		(*Delete SMS successfully executed*)
				EXIT;

			ELSIF	arDeleteSMSAnswerRcv[i]		= arAnswerErr[1]
				AND arDeleteSMSAnswerRcv[i+1] 	= arAnswerErr[2]
				AND arDeleteSMSAnswerRcv[i+2] 	= arAnswerErr[3]
				AND arDeleteSMSAnswerRcv[i+3] 	= arAnswerErr[4]
				AND arDeleteSMSAnswerRcv[i+4] 	= arAnswerErr[5]	THEN
					uiAnalyzeAnswer:=2;		(*Delete SMS failed*)
				EXIT;
			END_IF
		END_FOR

		CASE uiAnalyzeAnswer OF
			0:(*Undefined Answer*)
				bError:= TRUE;
				nErrorID:= 16#8010;
				nStep:=1000;

			1:(*Delete SMS successfully executed*)
				nStep:=1000;

			2:(*Delete SMS failed*)
				bError:= TRUE;
				nErrorID:= 16#800F;
				nStep:=1000;
		END_CASE


	900:(*Timeout*)
		bError:= TRUE;
		nErrorID:= 16#8001;
		nStep:=1000;


	1000:(*Reset Receive-FB*)
		fbReceiveData(	Reset:=TRUE,RXbuffer:= stRxBuffer);
		tonWaitTime(IN:=TRUE, PT:=t#500ms);
		IF	tonWaitTime.Q	THEN
			fbReceiveData(	Reset:=FALSE,RXbuffer:= stRxBuffer);
			nStep:=1010;
		END_IF


	1010:(*Send/Receive successful -> Reset FBs*)
		fbClearComBuffer(buffer:=stRxBuffer);
		fbClearComBuffer(buffer:=stTxBuffer);
		nStep:=0;
		bBusy:=FALSE;

	END_CASE;

END_FUNCTION_BLOCK

// ---- 00_FunctionsBlocks/Beckhoff/Communication/SMS/FB_Login.TcPOU
FUNCTION_BLOCK FB_Login

VAR_INPUT
	bStart					: BOOL;
	
END_VAR
VAR_OUTPUT
	bBusy					: BOOL;
	bError					: BOOL;
	nErrorID				: UINT;
END_VAR

VAR_IN_OUT
	stTxBuffer				: ComBuffer;
	stRxBuffer				: ComBuffer;
END_VAR

VAR
	rtrigStart				: R_TRIG;

	fbSendData				: SendData;
	fbReceiveData			: ReceiveData;
	fbClearComBuffer		: ClearComBuffer;

	i						: UINT;
	nStep					: UINT; (* sequence state *)
	tonWaitTime				: TON;
	tonTimeOut				: TON;
	tTimeout				: TIME:=t#30s;

	arAnswerOK				: ARRAY[1..2] OF BYTE:=[16#4F,16#4B];
	arAnswerErr				: ARRAY[1..5] OF BYTE:=[16#45,16#52,16#52,16#4F,16#52];

	sEchoOff				: STRING(5);			(*Command-String*)
	arEchoOff				: ARRAY[1..5] OF BYTE;	(*Command-ARRAY*)
	arEchoOffAnswerRcv		: ARRAY[1..5] OF BYTE;	(*Received answer of the command*)
	arEchoOffAnswerClr		: ARRAY[1..5] OF BYTE;	(*Empty-ARRAY to clear the answer for debugging*)

	sLogin					: STRING(21);			(*Command-String*)
	arLogin					: ARRAY[1..21] OF BYTE;	(*Command-ARRAY*)
	arLoginAnswerRcv		: ARRAY[1..5] OF BYTE;	(*Received answer of the command*)
	arLoginAnswerClr		: ARRAY[1..5] OF BYTE;	(*Empty-ARRAY to clear the answer for debugging*)
END_VAR

	rtrigStart(CLK:=bStart);  //Rising Edge detect

	tonTimeout();
	IF (tonTimeout.Q) THEN
		tonTimeout(IN := FALSE);
		nStep := 900;
	END_IF


	CASE nStep OF

	0: 	(*Idle Step*);
		tonTimeout(IN:=FALSE);
		tonWaitTime(IN:=FALSE);
		IF (rtrigStart.Q AND NOT bBusy) THEN
			nStep := 5;
			bBusy := TRUE;
		ELSE
			bBusy := FALSE;
		END_IF


	5:
		bError				:= FALSE;
		nErrorId			:= 0;
		tonTimeout			(IN := TRUE, PT := tTimeout);
		fbClearComBuffer	(buffer:=stRxBuffer);
		fbClearComBuffer	(buffer:=stTxBuffer);
		arEchoOffAnswerRcv	:= arEchoOffAnswerClr;
		arLoginAnswerRcv	:= arLoginAnswerClr;
	//	MEMSET(ADR(sMessageText),0,SIZEOF(sMessageText));
		nStep := 50;


	(*10:(*Length PIN-number within range?*)
		IF 		LEN(sPinNumber) < 1
			OR	LEN(sPinNumber) > 10 THEN
			bError		:= TRUE;
			nErrorID	:= 16#8002;
			nStep		:= 1000;
		ELSE
			nStep		:= 20;
		END_IF


	20:(*Phone-number contains correct characters? 0..9*)
		FOR i:=1 TO LEN(sPinNumber) DO
			IF 		ASC(MID(sPinNumber,1,i)) < 16#30
				OR	ASC(MID(sPinNumber,1,i)) > 16#39	(*a non-numeric character in PIN*)	THEN
				bError		:= TRUE;
				nErrorID	:= 16#8003;
			END_IF
		END_FOR

		IF bError	THEN
			nStep	:= 1000;
		ELSE
			nStep	:= 50;
		END_IF*)


	50:(*Create command-Arrays*)

